LIN {X 0,Y 466.782,Z 446.473,A -85,B 0,C 180,E1 -7483.052,E2 -7483.052} C_VEL
LIN {X 0,Y 466.617,Z 450.017,A -85,B 0,C 180,E1 -7484.835,E2 -7484.835} C_VEL
LIN {X 0,Y 466.515,Z 452.31,A -85,B 0,C 180,E1 -7486.632,E2 -7486.632} C_VEL
LIN {X 0,Y 466.556,Z 453.367,A -85,B 0,C 180,E1 -7488.441,E2 -7488.441} C_VEL
LIN {X 0,Y 466.556,Z 453.179,A -85,B 0,C 180,E1 -7490.271,E2 -7490.271} C_VEL
LIN {X 0,Y 466.538,Z 451.697,A -85,B 0,C 180,E1 -7492.123,E2 -7492.123} C_VEL
LIN {X 0,Y 466.702,Z 448.846,A -85,B 0,C 180,E1 -7493.99,E2 -7493.99} C_VEL
LIN {X 0,Y 466.897,Z 444.505,A -85,B 0,C 180,E1 -7495.882,E2 -7495.882} C_VEL
LIN {X 0,Y 467.049,Z 439.911,A -85,B 0,C 180,E1 -7497.399,E2 -7497.399} C_VEL
LIN {X 0,Y 467.44,Z 432.616,A -85,B 0,C 180,E1 -7499.303,E2 -7499.303} C_VEL
LIN {X 0,Y 467.943,Z 424.827,A -85,B 0,C 180,E1 -7500.924,E2 -7500.924} C_VEL
LIN {X 0,Y 468.484,Z 416.084,A -85,B 0,C 180,E1 -7502.432,E2 -7502.432} C_VEL
LIN {X 0,Y 469.232,Z 405.809,A -85,B 0,C 180,E1 -7503.912,E2 -7503.912} C_VEL
LIN {X 0,Y 469.994,Z 394.444,A -85,B 0,C 180,E1 -7505.28,E2 -7505.28} C_VEL
LIN {X 0,Y 470.915,Z 381.942,A -85,B 0,C 180,E1 -7506.527,E2 -7506.527} C_VEL
LIN {X 0,Y 471.73,Z 369.989,A -85,B 0,C 180,E1 -7507.515,E2 -7507.515} C_VEL
LIN {X 0,Y 472.515,Z 356.993,A -85,B 0,C 180,E1 -7508.405,E2 -7508.405} C_VEL
LIN {X 0,Y 473.293,Z 342.587,A -85,B 0,C 180,E1 -7509.192,E2 -7509.192} C_VEL
LIN {X 0,Y 473.911,Z 327.391,A -85,B 0,C 180,E1 -7509.826,E2 -7509.826} C_VEL
LIN {X 0,Y 474.427,Z 311.981,A -85,B 0,C 180,E1 -7510.276,E2 -7510.276} C_VEL
LIN {X 0,Y 474.73,Z 291.402,A -85,B 0,C 180,E1 -7510.646,E2 -7510.646} C_VEL
LIN {X 0,Y 476.309,Z 163.823,A -85,B 0,C 180,E1 -7512.654,E2 -7512.654} C_VEL
LIN {X 0,Y 472.095,Z 146.225,A -85,B 0,C 180,E1 -7513.196,E2 -7513.196} C_VEL
LIN {X 0,Y 471.241,Z 143.803,A -85,B 0,C 180,E1 -7513.317,E2 -7513.317} C_VEL
LIN {X 0,Y 468.712,Z 132.548,A -85,B 0,C 180,E1 -7515.49,E2 -7515.49} C_VEL
LIN {X 0,Y 467.569,Z 127.869,A -85,B 0,C 180,E1 -7516.442,E2 -7516.442} C_VEL
LIN {X 0,Y 467.571,Z 127.872,A -85,B 0,C 180,E1 -7519.734,E2 -7519.734} C_VEL
LIN {X 0,Y 467.544,Z 127.872,A -85,B 0,C 180,E1 -7522.814,E2 -7522.814} C_VEL
LIN {X 0,Y 467.588,Z 127.867,A -85,B 0,C 180,E1 -7526.211,E2 -7526.211} C_VEL
LIN {X 0,Y 467.57,Z 127.865,A -85,B 0,C 180,E1 -7529.266,E2 -7529.266} C_VEL
LIN {X 0,Y 467.605,Z 127.861,A -85,B 0,C 180,E1 -7532.468,E2 -7532.468} C_VEL
LIN {X 0,Y 467.569,Z 127.862,A -85,B 0,C 180,E1 -7535.11,E2 -7535.11} C_VEL
LIN {X 0,Y 467.536,Z 127.873,A -85,B 0,C 180,E1 -7537.926,E2 -7537.926} C_VEL
LIN {X 0,Y 467.622,Z 127.859,A -85,B 0,C 180,E1 -7540.692,E2 -7540.692} C_VEL
LIN {X 0,Y 467.639,Z 127.856,A -85,B 0,C 180,E1 -7544.305,E2 -7544.305} C_VEL
LIN {X 0,Y 467.657,Z 127.855,A -85,B 0,C 180,E1 -7547.854,E2 -7547.854} C_VEL
LIN {X 0,Y 467.681,Z 127.852,A -85,B 0,C 180,E1 -7551.357,E2 -7551.357} C_VEL
LIN {X 0,Y 467.735,Z 127.842,A -85,B 0,C 180,E1 -7553.962,E2 -7553.962} C_VEL
LIN {X 0,Y 467.859,Z 127.831,A -85,B 0,C 180,E1 -7557.417,E2 -7557.417} C_VEL
LIN {X 0,Y 467.883,Z 127.826,A -85,B 0,C 180,E1 -7560,E2 -7560} C_VEL
LIN {X 0,Y 467.859,Z 127.827,A -85,B 0,C 180,E1 -7562.583,E2 -7562.583} C_VEL
LIN {X 0,Y 467.724,Z 127.844,A -85,B 0,C 180,E1 -7566.037,E2 -7566.037} C_VEL
LIN {X 0,Y 467.659,Z 127.856,A -85,B 0,C 180,E1 -7569.515,E2 -7569.515} C_VEL
LIN {X 0,Y 467.654,Z 127.852,A -85,B 0,C 180,E1 -7572.357,E2 -7572.357} C_VEL
LIN {X 0,Y 467.649,Z 127.85,A -85,B 0,C 180,E1 -7575.885,E2 -7575.885} C_VEL
LIN {X 0,Y 467.621,Z 127.857,A -85,B 0,C 180,E1 -7579.308,E2 -7579.308} C_VEL
LIN {X 0,Y 467.534,Z 127.869,A -85,B 0,C 180,E1 -7582.074,E2 -7582.074} C_VEL
LIN {X 0,Y 467.594,Z 127.866,A -85,B 0,C 180,E1 -7584.888,E2 -7584.888} C_VEL
LIN {X 0,Y 467.619,Z 127.859,A -85,B 0,C 180,E1 -7587.769,E2 -7587.769} C_VEL
LIN {X 0,Y 467.567,Z 127.866,A -85,B 0,C 180,E1 -7591.045,E2 -7591.045} C_VEL
LIN {X 0,Y 467.575,Z 127.868,A -85,B 0,C 180,E1 -7594.24,E2 -7594.24} C_VEL
LIN {X 0,Y 467.546,Z 127.866,A -85,B 0,C 180,E1 -7597.186,E2 -7597.186} C_VEL
LIN {X 0,Y 467.573,Z 127.866,A -85,B 0,C 180,E1 -7600.265,E2 -7600.265} C_VEL
LIN {X 0,Y 467.585,Z 127.858,A -85,B 0,C 180,E1 -7602.567,E2 -7602.567} C_VEL
LIN {X 0,Y 467.569,Z 127.866,A -85,B 0,C 180,E1 -7605.053,E2 -7605.053} C_VEL
LIN {X 0,Y 467.587,Z 127.86,A -85,B 0,C 180,E1 -7607.44,E2 -7607.44} C_VEL
LIN {X 0,Y 467.581,Z 127.866,A -85,B 0,C 180,E1 -7610.855,E2 -7610.855} C_VEL
LIN {X 0,Y 467.558,Z 127.87,A -85,B 0,C 180,E1 -7614.261,E2 -7614.261} C_VEL
LIN {X 0,Y 467.58,Z 127.863,A -85,B 0,C 180,E1 -7617.321,E2 -7617.321} C_VEL
LIN {X 0,Y 467.597,Z 127.89,A -85,B 0,C 180,E1 -7619.394,E2 -7619.394} C_VEL
LIN {X 0,Y 471.135,Z 142.057,A -85,B 0,C 180,E1 -7621.918,E2 -7621.918} C_VEL
LIN {X 0,Y 472.352,Z 148.297,A -85,B 0,C 180,E1 -7622.972,E2 -7622.972} C_VEL
LIN {X 0,Y 471.282,Z 166.846,A -85,B 0,C 180,E1 -7625.75,E2 -7625.75} C_VEL
LIN {X 0,Y 476.101,Z 191.193,A -85,B 0,C 180,E1 -7626.44,E2 -7626.44} C_VEL
LIN {X 0,Y 474.313,Z 333.167,A -85,B 0,C 180,E1 -7628.686,E2 -7628.686} C_VEL
LIN {X 0,Y 473.716,Z 349.25,A -85,B 0,C 180,E1 -7629.113,E2 -7629.113} C_VEL
LIN {X 0,Y 473.056,Z 364.395,A -85,B 0,C 180,E1 -7629.704,E2 -7629.704} C_VEL
LIN {X 0,Y 472.265,Z 378.653,A -85,B 0,C 180,E1 -7630.438,E2 -7630.438} C_VEL
LIN {X 0,Y 471.44,Z 392.03,A -85,B 0,C 180,E1 -7631.306,E2 -7631.306} C_VEL
LIN {X 0,Y 470.527,Z 405.676,A -85,B 0,C 180,E1 -7632.395,E2 -7632.395} C_VEL
LIN {X 0,Y 469.658,Z 418.059,A -85,B 0,C 180,E1 -7633.594,E2 -7633.594} C_VEL
LIN {X 0,Y 468.795,Z 430.236,A -85,B 0,C 180,E1 -7635.013,E2 -7635.013} C_VEL
LIN {X 0,Y 468.095,Z 441.083,A -85,B 0,C 180,E1 -7636.543,E2 -7636.543} C_VEL
LIN {X 0,Y 467.588,Z 450.127,A -85,B 0,C 180,E1 -7638.073,E2 -7638.073} C_VEL
LIN {X 0,Y 467.221,Z 457.636,A -85,B 0,C 180,E1 -7639.601,E2 -7639.601} C_VEL
LIN {X 0,Y 466.904,Z 464.643,A -85,B 0,C 180,E1 -7641.343,E2 -7641.343} C_VEL
LIN {X 0,Y 466.742,Z 470.157,A -85,B 0,C 180,E1 -7643.082,E2 -7643.082} C_VEL
LIN {X 0,Y 466.684,Z 474.33,A -85,B 0,C 180,E1 -7644.816,E2 -7644.816} C_VEL
LIN {X 0,Y 466.634,Z 477.256,A -85,B 0,C 180,E1 -7646.546,E2 -7646.546} C_VEL
LIN {X 0,Y 466.604,Z 479.003,A -85,B 0,C 180,E1 -7648.274,E2 -7648.274} C_VEL
LIN {X 0,Y 466.596,Z 479.604,A -85,B 0,C 180,E1 -7650,E2 -7650} C_VEL
LIN {X 0,Y 466.604,Z 479.005,A -85,B 0,C 180,E1 -7651.727,E2 -7651.727} C_VEL
LIN {X 0,Y 466.634,Z 477.252,A -85,B 0,C 180,E1 -7653.454,E2 -7653.454} C_VEL
LIN {X 0,Y 466.686,Z 474.32,A -85,B 0,C 180,E1 -7655.184,E2 -7655.184} C_VEL
LIN {X 0,Y 466.818,Z 470.137,A -85,B 0,C 180,E1 -7656.918,E2 -7656.918} C_VEL
LIN {X 0,Y 466.906,Z 464.586,A -85,B 0,C 180,E1 -7658.658,E2 -7658.658} C_VEL
LIN {X 0,Y 467.225,Z 457.523,A -85,B 0,C 180,E1 -7660.4,E2 -7660.4} C_VEL
LIN {X 0,Y 467.608,Z 449.968,A -85,B 0,C 180,E1 -7661.927,E2 -7661.927} C_VEL
LIN {X 0,Y 468.072,Z 440.853,A -85,B 0,C 180,E1 -7663.458,E2 -7663.458} C_VEL
LIN {X 0,Y 468.787,Z 429.87,A -85,B 0,C 180,E1 -7664.988,E2 -7664.988} C_VEL
LIN {X 0,Y 469.549,Z 418.573,A -85,B 0,C 180,E1 -7666.299,E2 -7666.299} C_VEL
LIN {X 0,Y 470.358,Z 406.169,A -85,B 0,C 180,E1 -7667.5,E2 -7667.5} C_VEL
LIN {X 0,Y 471.26,Z 392.481,A -85,B 0,C 180,E1 -7668.589,E2 -7668.589} C_VEL
LIN {X 0,Y 472.067,Z 379.034,A -85,B 0,C 180,E1 -7669.458,E2 -7669.458} C_VEL
LIN {X 0,Y 472.869,Z 364.303,A -85,B 0,C 180,E1 -7670.212,E2 -7670.212} C_VEL
LIN {X 0,Y 473.486,Z 349.003,A -85,B 0,C 180,E1 -7670.8,E2 -7670.8} C_VEL
LIN {X 0,Y 473.96,Z 333.066,A -85,B 0,C 180,E1 -7671.218,E2 -7671.218} C_VEL
LIN {X 0,Y 475.74,Z 191.939,A -85,B 0,C 180,E1 -7673.418,E2 -7673.418} C_VEL
LIN {X 0,Y 471.033,Z 167.135,A -85,B 0,C 180,E1 -7674.068,E2 -7674.068} C_VEL
LIN {X 0,Y 472.031,Z 148.627,A -85,B 0,C 180,E1 -7676.782,E2 -7676.782} C_VEL
LIN {X 0,Y 471.422,Z 143.906,A -85,B 0,C 180,E1 -7677.526,E2 -7677.526} C_VEL
LIN {X 0,Y 467.57,Z 127.869,A -85,B 0,C 180,E1 -7680.235,E2 -7680.235} C_VEL
LIN {X 0,Y 467.585,Z 127.868,A -85,B 0,C 180,E1 -7682.759,E2 -7682.759} C_VEL
LIN {X 0,Y 467.555,Z 127.873,A -85,B 0,C 180,E1 -7685.89,E2 -7685.89} C_VEL
LIN {X 0,Y 467.56,Z 127.867,A -85,B 0,C 180,E1 -7689.148,E2 -7689.148} C_VEL
LIN {X 0,Y 467.575,Z 127.868,A -85,B 0,C 180,E1 -7691.404,E2 -7691.404} C_VEL
LIN {X 0,Y 467.568,Z 127.868,A -85,B 0,C 180,E1 -7695.053,E2 -7695.053} C_VEL
LIN {X 0,Y 467.591,Z 127.87,A -85,B 0,C 180,E1 -7697.44,E2 -7697.44} C_VEL
LIN {X 0,Y 467.561,Z 127.864,A -85,B 0,C 180,E1 -7700.853,E2 -7700.853} C_VEL
LIN {X 0,Y 467.562,Z 127.864,A -85,B 0,C 180,E1 -7704.262,E2 -7704.262} C_VEL
LIN {X 0,Y 467.582,Z 127.867,A -85,B 0,C 180,E1 -7707.322,E2 -7707.322} C_VEL
LIN {X 0,Y 467.545,Z 127.865,A -85,B 0,C 180,E1 -7710.262,E2 -7710.262} C_VEL
LIN {X 0,Y 467.566,Z 127.86,A -85,B 0,C 180,E1 -7713.197,E2 -7713.197} C_VEL
LIN {X 0,Y 467.593,Z 127.862,A -85,B 0,C 180,E1 -7716.47,E2 -7716.47} C_VEL
LIN {X 0,Y 467.625,Z 127.856,A -85,B 0,C 180,E1 -7719.778,E2 -7719.778} C_VEL
LIN {X 0,Y 467.597,Z 127.864,A -85,B 0,C 180,E1 -7722.507,E2 -7722.507} C_VEL
LIN {X 0,Y 467.6,Z 127.862,A -85,B 0,C 180,E1 -7725.197,E2 -7725.197} C_VEL
LIN {X 0,Y 467.661,Z 127.85,A -85,B 0,C 180,E1 -7727.855,E2 -7727.855} C_VEL
LIN {X 0,Y 467.668,Z 127.85,A -85,B 0,C 180,E1 -7731.357,E2 -7731.357} C_VEL
LIN {X 0,Y 467.706,Z 127.848,A -85,B 0,C 180,E1 -7733.962,E2 -7733.962} C_VEL
LIN {X 0,Y 467.817,Z 127.828,A -85,B 0,C 180,E1 -7737.417,E2 -7737.417} C_VEL
LIN {X 0,Y 467.853,Z 127.817,A -85,B 0,C 180,E1 -7740,E2 -7740} C_VEL
LIN {X 0,Y 467.815,Z 127.833,A -85,B 0,C 180,E1 -7742.584,E2 -7742.584} C_VEL
LIN {X 0,Y 467.705,Z 127.85,A -85,B 0,C 180,E1 -7746.038,E2 -7746.038} C_VEL
LIN {X 0,Y 467.634,Z 127.842,A -85,B 0,C 180,E1 -7748.644,E2 -7748.644} C_VEL
LIN {X 0,Y 467.646,Z 127.855,A -85,B 0,C 180,E1 -7752.146,E2 -7752.146} C_VEL
LIN {X 0,Y 467.582,Z 127.867,A -85,B 0,C 180,E1 -7755.697,E2 -7755.697} C_VEL
LIN {X 0,Y 467.553,Z 127.865,A -85,B 0,C 180,E1 -7758.739,E2 -7758.739} C_VEL
LIN {X 0,Y 467.517,Z 127.869,A -85,B 0,C 180,E1 -7762.075,E2 -7762.075} C_VEL
LIN {X 0,Y 467.531,Z 127.87,A -85,B 0,C 180,E1 -7764.892,E2 -7764.892} C_VEL
LIN {X 0,Y 467.542,Z 127.86,A -85,B 0,C 180,E1 -7767.775,E2 -7767.775} C_VEL
LIN {X 0,Y 467.532,Z 127.862,A -85,B 0,C 180,E1 -7771.036,E2 -7771.036} C_VEL
LIN {X 0,Y 467.568,Z 127.863,A -85,B 0,C 180,E1 -7774.238,E2 -7774.238} C_VEL
LIN {X 0,Y 467.518,Z 127.863,A -85,B 0,C 180,E1 -7777.181,E2 -7777.181} C_VEL
LIN {X 0,Y 467.561,Z 127.861,A -85,B 0,C 180,E1 -7780.267,E2 -7780.267} C_VEL
LIN {X 0,Y 467.55,Z 127.864,A -85,B 0,C 180,E1 -7783.746,E2 -7783.746} C_VEL
LIN {X 0,Y 467.55,Z 127.857,A -85,B 0,C 180,E1 -7786.254,E2 -7786.254} C_VEL
LIN {X 0,Y 467.561,Z 127.865,A -85,B 0,C 180,E1 -7789.733,E2 -7789.733} C_VEL
LIN {X 0,Y 467.526,Z 127.869,A -85,B 0,C 180,E1 -7793.037,E2 -7793.037} C_VEL
LIN {X 0,Y 467.573,Z 127.868,A -85,B 0,C 180,E1 -7796.21,E2 -7796.21} C_VEL
LIN {X 0,Y 467.571,Z 127.865,A -85,B 0,C 180,E1 -7799.266,E2 -7799.266} C_VEL
LIN {X 0,Y 467.556,Z 127.872,A -85,B 0,C 180,E1 -7802.481,E2 -7802.481} C_VEL
LIN {X 0,Y 467.565,Z 127.867,A -85,B 0,C 180,E1 -7805.11,E2 -7805.11} C_VEL
LIN {X 0,Y 467.54,Z 127.874,A -85,B 0,C 180,E1 -7807.926,E2 -7807.926} C_VEL
LIN {X 0,Y 467.626,Z 127.856,A -85,B 0,C 180,E1 -7810.692,E2 -7810.692} C_VEL
LIN {X 0,Y 467.644,Z 127.859,A -85,B 0,C 180,E1 -7814.305,E2 -7814.305} C_VEL
LIN {X 0,Y 467.598,Z 127.861,A -85,B 0,C 180,E1 -7815.378,E2 -7815.378} C_VEL
LIN {X 0,Y 466.926,Z 127.942,A -85,B 0,C 180,E1 -7816.097,E2 -7816.097} C_VEL
LIN {X 0,Y 464.087,Z 128.299,A -85,B 0,C 180,E1 -7817.265,E2 -7817.265} C_VEL
LIN {X 0,Y 461.69,Z 128.601,A -85,B 0,C 180,E1 -7818.208,E2 -7818.208} C_VEL
LIN {X 0,Y 460.662,Z 128.729,A -85,B 0,C 180,E1 -7818.936,E2 -7818.936} C_VEL
LIN {X 0,Y 460.578,Z 128.74,A -85,B 0,C 180,E1 -7819.182,E2 -7819.182} C_VEL
LIN {X 0,Y 460.666,Z 128.88,A -85,B 0,C 180,E1 -7821.832,E2 -7821.832} C_VEL
LIN {X 0,Y 463.902,Z 143.363,A -85,B 0,C 180,E1 -7824.566,E2 -7824.566} C_VEL
LIN {X 0,Y 463.975,Z 143.816,A -85,B 0,C 180,E1 -7824.649,E2 -7824.649} C_VEL
LIN {X 0,Y 465.945,Z 150.272,A -85,B 0,C 180,E1 -7824.861,E2 -7824.861} C_VEL
LIN {X 0,Y 469.269,Z 165.031,A -85,B 0,C 180,E1 -7825.274,E2 -7825.274} C_VEL
LIN {X 0,Y 467.513,Z 308.285,A -85,B 0,C 180,E1 -7827.55,E2 -7827.55} C_VEL
LIN {X 0,Y 467.068,Z 323.449,A -85,B 0,C 180,E1 -7827.952,E2 -7827.952} C_VEL
LIN {X 0,Y 466.484,Z 338.755,A -85,B 0,C 180,E1 -7828.543,E2 -7828.543} C_VEL
LIN {X 0,Y 465.789,Z 352.417,A -85,B 0,C 180,E1 -7829.243,E2 -7829.243} C_VEL
LIN {X 0,Y 464.987,Z 365.876,A -85,B 0,C 180,E1 -7830.108,E2 -7830.108} C_VEL
LIN {X 0,Y 464.087,Z 378.978,A -85,B 0,C 180,E1 -7831.141,E2 -7831.141} C_VEL
LIN {X 0,Y 463.273,Z 390.919,A -85,B 0,C 180,E1 -7832.282,E2 -7832.282} C_VEL
LIN {X 0,Y 462.469,Z 401.527,A -85,B 0,C 180,E1 -7833.485,E2 -7833.485} C_VEL
LIN {X 0,Y 461.736,Z 411.376,A -85,B 0,C 180,E1 -7834.802,E2 -7834.802} C_VEL
LIN {X 0,Y 461.14,Z 421.006,A -85,B 0,C 180,E1 -7836.343,E2 -7836.343} C_VEL
LIN {X 0,Y 460.609,Z 429.084,A -85,B 0,C 180,E1 -7837.893,E2 -7837.893} C_VEL
LIN {X 0,Y 460.133,Z 436.655,A -85,B 0,C 180,E1 -7839.672,E2 -7839.672} C_VEL
LIN {X 0,Y 459.858,Z 442.694,A -85,B 0,C 180,E1 -7841.459,E2 -7841.459} C_VEL
LIN {X 0,Y 459.664,Z 447.348,A -85,B 0,C 180,E1 -7843.258,E2 -7843.258} C_VEL
LIN {X 0,Y 459.528,Z 450.686,A -85,B 0,C 180,E1 -7845.07,E2 -7845.07} C_VEL
LIN {X 0,Y 459.429,Z 452.771,A -85,B 0,C 180,E1 -7846.896,E2 -7846.896} C_VEL
LIN {X 0,Y 459.443,Z 453.621,A -85,B 0,C 180,E1 -7848.737,E2 -7848.737} C_VEL
LIN {X 0,Y 459.449,Z 453.22,A -85,B 0,C 180,E1 -7850.598,E2 -7850.598} C_VEL
LIN {X 0,Y 459.464,Z 451.518,A -85,B 0,C 180,E1 -7852.482,E2 -7852.482} C_VEL
LIN {X 0,Y 459.645,Z 448.435,A -85,B 0,C 180,E1 -7854.383,E2 -7854.383} C_VEL
LIN {X 0,Y 459.862,Z 443.845,A -85,B 0,C 180,E1 -7856.308,E2 -7856.308} C_VEL
LIN {X 0,Y 460.067,Z 438.9,A -85,B 0,C 180,E1 -7857.895,E2 -7857.895} C_VEL
LIN {X 0,Y 460.456,Z 432.522,A -85,B 0,C 180,E1 -7859.54,E2 -7859.54} C_VEL
LIN {X 0,Y 461.008,Z 424.517,A -85,B 0,C 180,E1 -7861.22,E2 -7861.22} C_VEL
LIN {X 0,Y 461.591,Z 415.894,A -85,B 0,C 180,E1 -7862.718,E2 -7862.718} C_VEL
LIN {X 0,Y 462.397,Z 405.555,A -85,B 0,C 180,E1 -7864.219,E2 -7864.219} C_VEL
LIN {X 0,Y 463.258,Z 394.112,A -85,B 0,C 180,E1 -7865.604,E2 -7865.604} C_VEL
LIN {X 0,Y 464.244,Z 381.493,A -85,B 0,C 180,E1 -7866.868,E2 -7866.868} C_VEL
LIN {X 0,Y 465.203,Z 367.754,A -85,B 0,C 180,E1 -7867.997,E2 -7867.997} C_VEL
LIN {X 0,Y 466.106,Z 353.975,A -85,B 0,C 180,E1 -7868.91,E2 -7868.91} C_VEL
LIN {X 0,Y 466.896,Z 339.006,A -85,B 0,C 180,E1 -7869.69,E2 -7869.69} C_VEL
LIN {X 0,Y 467.472,Z 324.137,A -85,B 0,C 180,E1 -7870.275,E2 -7870.275} C_VEL
LIN {X 0,Y 468.003,Z 308.311,A -85,B 0,C 180,E1 -7870.697,E2 -7870.697} C_VEL
LIN {X 0,Y 469.919,Z 165.105,A -85,B 0,C 180,E1 -7873.005,E2 -7873.005} C_VEL
LIN {X 0,Y 466.02,Z 148.879,A -85,B 0,C 180,E1 -7873.518,E2 -7873.518} C_VEL
LIN {X 0,Y 464.143,Z 144.12,A -85,B 0,C 180,E1 -7873.733,E2 -7873.733} C_VEL
LIN {X 0,Y 461.347,Z 132.074,A -85,B 0,C 180,E1 -7876.121,E2 -7876.121} C_VEL
LIN {X 0,Y 460.54,Z 128.745,A -85,B 0,C 180,E1 -7876.816,E2 -7876.816} C_VEL
LIN {X 0,Y 460.52,Z 128.748,A -85,B 0,C 180,E1 -7880.136,E2 -7880.136} C_VEL
LIN {X 0,Y 460.474,Z 128.752,A -85,B 0,C 180,E1 -7883.47,E2 -7883.47} C_VEL
LIN {X 0,Y 460.531,Z 128.744,A -85,B 0,C 180,E1 -7886.675,E2 -7886.675} C_VEL
LIN {X 0,Y 460.508,Z 128.747,A -85,B 0,C 180,E1 -7889.759,E2 -7889.759} C_VEL
LIN {X 0,Y 460.535,Z 128.741,A -85,B 0,C 180,E1 -7892.753,E2 -7892.753} C_VEL
LIN {X 0,Y 460.522,Z 128.738,A -85,B 0,C 180,E1 -7895.666,E2 -7895.666} C_VEL
LIN {X 0,Y 460.523,Z 128.743,A -85,B 0,C 180,E1 -7898.578,E2 -7898.578} C_VEL
LIN {X 0,Y 460.586,Z 128.737,A -85,B 0,C 180,E1 -7901.31,E2 -7901.31} C_VEL
LIN {X 0,Y 460.605,Z 128.734,A -85,B 0,C 180,E1 -7904.059,E2 -7904.059} C_VEL
LIN {X 0,Y 460.61,Z 128.734,A -85,B 0,C 180,E1 -7907.665,E2 -7907.665} C_VEL
LIN {X 0,Y 460.628,Z 128.73,A -85,B 0,C 180,E1 -7911.223,E2 -7911.223} C_VEL
LIN {X 0,Y 460.701,Z 128.719,A -85,B 0,C 180,E1 -7913.87,E2 -7913.87} C_VEL
LIN {X 0,Y 460.799,Z 128.711,A -85,B 0,C 180,E1 -7917.377,E2 -7917.377} C_VEL
LIN {X 0,Y 460.853,Z 128.702,A -85,B 0,C 180,E1 -7920,E2 -7920} C_VEL
LIN {X 0,Y 460.8,Z 128.706,A -85,B 0,C 180,E1 -7922.622,E2 -7922.622} C_VEL
LIN {X 0,Y 460.688,Z 128.721,A -85,B 0,C 180,E1 -7926.13,E2 -7926.13} C_VEL
LIN {X 0,Y 460.619,Z 128.731,A -85,B 0,C 180,E1 -7928.776,E2 -7928.776} C_VEL
LIN {X 0,Y 460.613,Z 128.729,A -85,B 0,C 180,E1 -7932.445,E2 -7932.445} C_VEL
LIN {X 0,Y 460.6,Z 128.728,A -85,B 0,C 180,E1 -7935.997,E2 -7935.997} C_VEL
LIN {X 0,Y 460.567,Z 128.734,A -85,B 0,C 180,E1 -7939.615,E2 -7939.615} C_VEL
LIN {X 0,Y 460.51,Z 128.747,A -85,B 0,C 180,E1 -7942.428,E2 -7942.428} C_VEL
LIN {X 0,Y 460.557,Z 128.736,A -85,B 0,C 180,E1 -7945.799,E2 -7945.799} C_VEL
LIN {X 0,Y 460.551,Z 128.742,A -85,B 0,C 180,E1 -7948.233,E2 -7948.233} C_VEL
LIN {X 0,Y 460.519,Z 128.743,A -85,B 0,C 180,E1 -7951.283,E2 -7951.283} C_VEL
LIN {X 0,Y 460.521,Z 128.746,A -85,B 0,C 180,E1 -7954.504,E2 -7954.504} C_VEL
LIN {X 0,Y 460.499,Z 128.743,A -85,B 0,C 180,E1 -7957.623,E2 -7957.623} C_VEL
LIN {X 0,Y 460.537,Z 128.742,A -85,B 0,C 180,E1 -7960.269,E2 -7960.269} C_VEL
LIN {X 0,Y 460.498,Z 128.738,A -85,B 0,C 180,E1 -7963.375,E2 -7963.375} C_VEL
LIN {X 0,Y 460.498,Z 128.742,A -85,B 0,C 180,E1 -7966.625,E2 -7966.625} C_VEL
LIN {X 0,Y 460.54,Z 128.74,A -85,B 0,C 180,E1 -7969.731,E2 -7969.731} C_VEL
LIN {X 0,Y 460.498,Z 128.745,A -85,B 0,C 180,E1 -7972.524,E2 -7972.524} C_VEL
LIN {X 0,Y 460.545,Z 128.741,A -85,B 0,C 180,E1 -7975.624,E2 -7975.624} C_VEL
LIN {X 0,Y 460.531,Z 128.762,A -85,B 0,C 180,E1 -7979,E2 -7979} C_VEL
LIN {X 0,Y 463.991,Z 142.229,A -85,B 0,C 180,E1 -7981.464,E2 -7981.464} C_VEL
LIN {X 0,Y 465.574,Z 150.285,A -85,B 0,C 180,E1 -7982.855,E2 -7982.855} C_VEL
LIN {X 0,Y 464.571,Z 166.588,A -85,B 0,C 180,E1 -7985.338,E2 -7985.338} C_VEL
LIN {X 0,Y 469.673,Z 192.497,A -85,B 0,C 180,E1 -7986.096,E2 -7986.096} C_VEL
LIN {X 0,Y 467.74,Z 333.751,A -85,B 0,C 180,E1 -7988.371,E2 -7988.371} C_VEL
LIN {X 0,Y 467.106,Z 349.529,A -85,B 0,C 180,E1 -7988.804,E2 -7988.804} C_VEL
LIN {X 0,Y 466.384,Z 364.91,A -85,B 0,C 180,E1 -7989.42,E2 -7989.42} C_VEL
LIN {X 0,Y 465.583,Z 378.735,A -85,B 0,C 180,E1 -7990.145,E2 -7990.145} C_VEL
LIN {X 0,Y 464.691,Z 392.073,A -85,B 0,C 180,E1 -7991.025,E2 -7991.025} C_VEL
LIN {X 0,Y 463.717,Z 405.668,A -85,B 0,C 180,E1 -7992.127,E2 -7992.127} C_VEL
LIN {X 0,Y 462.8,Z 418.02,A -85,B 0,C 180,E1 -7993.344,E2 -7993.344} C_VEL
LIN {X 0,Y 461.887,Z 430.143,A -85,B 0,C 180,E1 -7994.783,E2 -7994.783} C_VEL
LIN {X 0,Y 461.113,Z 440.953,A -85,B 0,C 180,E1 -7996.335,E2 -7996.335} C_VEL
LIN {X 0,Y 460.571,Z 449.974,A -85,B 0,C 180,E1 -7997.889,E2 -7997.889} C_VEL
LIN {X 0,Y 460.208,Z 457.479,A -85,B 0,C 180,E1 -7999.441,E2 -7999.441} C_VEL
LIN {X 0,Y 459.847,Z 464.478,A -85,B 0,C 180,E1 -8001.209,E2 -8001.209} C_VEL
LIN {X 0,Y 459.662,Z 469.985,A -85,B 0,C 180,E1 -8002.975,E2 -8002.975} C_VEL
LIN {X 0,Y 459.595,Z 474.15,A -85,B 0,C 180,E1 -8004.736,E2 -8004.736} C_VEL
LIN {X 0,Y 459.529,Z 477.07,A -85,B 0,C 180,E1 -8006.493,E2 -8006.493} C_VEL
LIN {X 0,Y 459.517,Z 478.81,A -85,B 0,C 180,E1 -8008.247,E2 -8008.247} C_VEL
LIN {X 0,Y 459.527,Z 479.405,A -85,B 0,C 180,E1 -8010,E2 -8010} C_VEL
LIN {X 0,Y 459.517,Z 478.8,A -85,B 0,C 180,E1 -8011.753,E2 -8011.753} C_VEL
LIN {X 0,Y 459.53,Z 477.038,A -85,B 0,C 180,E1 -8013.508,E2 -8013.508} C_VEL
LIN {X 0,Y 459.598,Z 474.096,A -85,B 0,C 180,E1 -8015.265,E2 -8015.265} C_VEL
LIN {X 0,Y 459.727,Z 469.902,A -85,B 0,C 180,E1 -8017.025,E2 -8017.025} C_VEL
LIN {X 0,Y 459.848,Z 464.339,A -85,B 0,C 180,E1 -8018.792,E2 -8018.792} C_VEL
LIN {X 0,Y 460.202,Z 457.264,A -85,B 0,C 180,E1 -8020.56,E2 -8020.56} C_VEL
LIN {X 0,Y 460.584,Z 449.695,A -85,B 0,C 180,E1 -8022.112,E2 -8022.112} C_VEL
LIN {X 0,Y 461.108,Z 440.568,A -85,B 0,C 180,E1 -8023.665,E2 -8023.665} C_VEL
LIN {X 0,Y 461.855,Z 429.56,A -85,B 0,C 180,E1 -8025.218,E2 -8025.218} C_VEL
LIN {X 0,Y 462.672,Z 418.234,A -85,B 0,C 180,E1 -8026.548,E2 -8026.548} C_VEL
LIN {X 0,Y 463.525,Z 405.778,A -85,B 0,C 180,E1 -8027.767,E2 -8027.767} C_VEL
LIN {X 0,Y 464.473,Z 392.009,A -85,B 0,C 180,E1 -8028.871,E2 -8028.871} C_VEL
LIN {X 0,Y 465.338,Z 378.488,A -85,B 0,C 180,E1 -8029.751,E2 -8029.751} C_VEL
LIN {X 0,Y 466.15,Z 364.121,A -85,B 0,C 180,E1 -8030.492,E2 -8030.492} C_VEL
LIN {X 0,Y 466.771,Z 349.319,A -85,B 0,C 180,E1 -8031.072,E2 -8031.072} C_VEL
LIN {X 0,Y 467.294,Z 333.178,A -85,B 0,C 180,E1 -8031.506,E2 -8031.506} C_VEL
LIN {X 0,Y 469.146,Z 192.736,A -85,B 0,C 180,E1 -8033.729,E2 -8033.729} C_VEL
LIN {X 0,Y 464.228,Z 166.936,A -85,B 0,C 180,E1 -8034.419,E2 -8034.419} C_VEL
LIN {X 0,Y 465.196,Z 149.867,A -85,B 0,C 180,E1 -8036.957,E2 -8036.957} C_VEL
LIN {X 0,Y 464.453,Z 145.092,A -85,B 0,C 180,E1 -8037.73,E2 -8037.73} C_VEL
LIN {X 0,Y 460.522,Z 128.748,A -85,B 0,C 180,E1 -8040.525,E2 -8040.525} C_VEL
LIN {X 0,Y 460.531,Z 128.748,A -85,B 0,C 180,E1 -8043.325,E2 -8043.325} C_VEL
LIN {X 0,Y 460.478,Z 128.753,A -85,B 0,C 180,E1 -8046.53,E2 -8046.53} C_VEL
LIN {X 0,Y 460.535,Z 128.742,A -85,B 0,C 180,E1 -8048.896,E2 -8048.896} C_VEL
LIN {X 0,Y 460.505,Z 128.747,A -85,B 0,C 180,E1 -8052.184,E2 -8052.184} C_VEL
LIN {X 0,Y 460.516,Z 128.751,A -85,B 0,C 180,E1 -8055.412,E2 -8055.412} C_VEL
LIN {X 0,Y 460.534,Z 128.743,A -85,B 0,C 180,E1 -8058.398,E2 -8058.398} C_VEL
LIN {X 0,Y 460.52,Z 128.742,A -85,B 0,C 180,E1 -8061.267,E2 -8061.267} C_VEL
LIN {X 0,Y 460.511,Z 128.742,A -85,B 0,C 180,E1 -8064.555,E2 -8064.555} C_VEL
LIN {X 0,Y 460.532,Z 128.742,A -85,B 0,C 180,E1 -8067.716,E2 -8067.716} C_VEL
LIN {X 0,Y 460.523,Z 128.743,A -85,B 0,C 180,E1 -8070.768,E2 -8070.768} C_VEL
LIN {X 0,Y 460.534,Z 128.735,A -85,B 0,C 180,E1 -8073.733,E2 -8073.733} C_VEL
LIN {X 0,Y 460.547,Z 128.742,A -85,B 0,C 180,E1 -8076.624,E2 -8076.624} C_VEL
LIN {X 0,Y 460.554,Z 128.738,A -85,B 0,C 180,E1 -8079.453,E2 -8079.453} C_VEL
LIN {X 0,Y 460.549,Z 128.739,A -85,B 0,C 180,E1 -8082.23,E2 -8082.23} C_VEL
LIN {X 0,Y 460.562,Z 128.741,A -85,B 0,C 180,E1 -8084.965,E2 -8084.965} C_VEL
LIN {X 0,Y 460.613,Z 128.734,A -85,B 0,C 180,E1 -8088.56,E2 -8088.56} C_VEL
LIN {X 0,Y 460.619,Z 128.728,A -85,B 0,C 180,E1 -8091.224,E2 -8091.224} C_VEL
LIN {X 0,Y 460.672,Z 128.723,A -85,B 0,C 180,E1 -8093.87,E2 -8093.87} C_VEL
LIN {X 0,Y 460.761,Z 128.707,A -85,B 0,C 180,E1 -8097.378,E2 -8097.378} C_VEL
LIN {X 0,Y 460.823,Z 128.692,A -85,B 0,C 180,E1 -8100,E2 -8100} C_VEL
LIN {X 0,Y 460.759,Z 128.712,A -85,B 0,C 180,E1 -8102.623,E2 -8102.623} C_VEL
LIN {X 0,Y 460.671,Z 128.724,A -85,B 0,C 180,E1 -8106.131,E2 -8106.131} C_VEL
LIN {X 0,Y 460.589,Z 128.718,A -85,B 0,C 180,E1 -8108.777,E2 -8108.777} C_VEL
LIN {X 0,Y 460.602,Z 128.73,A -85,B 0,C 180,E1 -8112.435,E2 -8112.435} C_VEL
LIN {X 0,Y 460.531,Z 128.741,A -85,B 0,C 180,E1 -8115.965,E2 -8115.965} C_VEL
LIN {X 0,Y 460.514,Z 128.742,A -85,B 0,C 180,E1 -8118.879,E2 -8118.879} C_VEL
LIN {X 0,Y 460.492,Z 128.742,A -85,B 0,C 180,E1 -8122.43,E2 -8122.43} C_VEL
LIN {X 0,Y 460.526,Z 128.742,A -85,B 0,C 180,E1 -8125.79,E2 -8125.79} C_VEL
LIN {X 0,Y 460.5,Z 128.734,A -85,B 0,C 180,E1 -8128.237,E2 -8128.237} C_VEL
LIN {X 0,Y 460.5,Z 128.741,A -85,B 0,C 180,E1 -8131.278,E2 -8131.278} C_VEL
LIN {X 0,Y 460.515,Z 128.743,A -85,B 0,C 180,E1 -8134.501,E2 -8134.501} C_VEL
LIN {X 0,Y 460.486,Z 128.734,A -85,B 0,C 180,E1 -8137.625,E2 -8137.625} C_VEL
LIN {X 0,Y 460.519,Z 128.747,A -85,B 0,C 180,E1 -8141.013,E2 -8141.013} C_VEL
LIN {X 0,Y 460.516,Z 128.743,A -85,B 0,C 180,E1 -8144.589,E2 -8144.589} C_VEL
LIN {X 0,Y 460.48,Z 128.745,A -85,B 0,C 180,E1 -8147.813,E2 -8147.813} C_VEL
LIN {X 0,Y 460.516,Z 128.745,A -85,B 0,C 180,E1 -8150.135,E2 -8150.135} C_VEL
LIN {X 0,Y 460.476,Z 128.745,A -85,B 0,C 180,E1 -8153.47,E2 -8153.47} C_VEL
LIN {X 0,Y 460.522,Z 128.74,A -85,B 0,C 180,E1 -8156.674,E2 -8156.674} C_VEL
LIN {X 0,Y 460.509,Z 128.746,A -85,B 0,C 180,E1 -8159.759,E2 -8159.759} C_VEL
LIN {X 0,Y 460.497,Z 128.749,A -85,B 0,C 180,E1 -8162.751,E2 -8162.751} C_VEL
LIN {X 0,Y 460.523,Z 128.746,A -85,B 0,C 180,E1 -8165.666,E2 -8165.666} C_VEL
LIN {X 0,Y 460.527,Z 128.744,A -85,B 0,C 180,E1 -8168.578,E2 -8168.578} C_VEL
LIN {X 0,Y 460.589,Z 128.733,A -85,B 0,C 180,E1 -8171.31,E2 -8171.31} C_VEL
LIN {X 0,Y 460.61,Z 128.738,A -85,B 0,C 180,E1 -8174.059,E2 -8174.059} C_VEL
LIN {X 0,Y 460.615,Z 128.736,A -85,B 0,C 180,E1 -8177.666,E2 -8177.666} C_VEL
LIN {X 0,Y 460.578,Z 128.74,A -85,B 0,C 180,E1 -8179.182,E2 -8179.182} C_VEL
LIN {X 0,Y 459.847,Z 128.893,A -85,B 0,C 180,E1 -8179.69,E2 -8179.69} C_VEL
LIN {X 0,Y 454.181,Z 129.586,A -85,B 0,C 180,E1 -8181.254,E2 -8181.254} C_VEL
LIN {X 0,Y 453.765,Z 130.303,A -85,B 0,C 180,E1 -8181.633,E2 -8181.633} C_VEL
LIN {X 0,Y 453.816,Z 130.602,A -85,B 0,C 180,E1 -8181.702,E2 -8181.702} C_VEL
LIN {X 0,Y 456.858,Z 144.007,A -85,B 0,C 180,E1 -8184.271,E2 -8184.271} C_VEL
LIN {X 0,Y 459.358,Z 151.363,A -85,B 0,C 180,E1 -8184.532,E2 -8184.532} C_VEL
LIN {X 0,Y 462.738,Z 166.534,A -85,B 0,C 180,E1 -8184.964,E2 -8184.964} C_VEL
LIN {X 0,Y 460.817,Z 309.517,A -85,B 0,C 180,E1 -8187.268,E2 -8187.268} C_VEL
LIN {X 0,Y 460.338,Z 325.111,A -85,B 0,C 180,E1 -8187.703,E2 -8187.703} C_VEL
LIN {X 0,Y 459.754,Z 339.99,A -85,B 0,C 180,E1 -8188.302,E2 -8188.302} C_VEL
LIN {X 0,Y 459.023,Z 353.474,A -85,B 0,C 180,E1 -8189.013,E2 -8189.013} C_VEL
LIN {X 0,Y 458.174,Z 366.768,A -85,B 0,C 180,E1 -8189.89,E2 -8189.89} C_VEL
LIN {X 0,Y 457.21,Z 380.349,A -85,B 0,C 180,E1 -8190.991,E2 -8190.991} C_VEL
LIN {X 0,Y 456.26,Z 392.664,A -85,B 0,C 180,E1 -8192.207,E2 -8192.207} C_VEL
LIN {X 0,Y 455.421,Z 403.883,A -85,B 0,C 180,E1 -8193.539,E2 -8193.539} C_VEL
LIN {X 0,Y 454.676,Z 413.378,A -85,B 0,C 180,E1 -8194.877,E2 -8194.877} C_VEL
LIN {X 0,Y 454.051,Z 422.718,A -85,B 0,C 180,E1 -8196.443,E2 -8196.443} C_VEL
LIN {X 0,Y 453.531,Z 430.532,A -85,B 0,C 180,E1 -8198.017,E2 -8198.017} C_VEL
LIN {X 0,Y 453.016,Z 437.873,A -85,B 0,C 180,E1 -8199.825,E2 -8199.825} C_VEL
LIN {X 0,Y 452.774,Z 443.682,A -85,B 0,C 180,E1 -8201.641,E2 -8201.641} C_VEL
LIN {X 0,Y 452.534,Z 448.128,A -85,B 0,C 180,E1 -8203.471,E2 -8203.471} C_VEL
LIN {X 0,Y 452.431,Z 451.282,A -85,B 0,C 180,E1 -8205.312,E2 -8205.312} C_VEL
LIN {X 0,Y 452.325,Z 453.205,A -85,B 0,C 180,E1 -8207.17,E2 -8207.17} C_VEL
LIN {X 0,Y 452.343,Z 453.875,A -85,B 0,C 180,E1 -8209.043,E2 -8209.043} C_VEL
LIN {X 0,Y 452.373,Z 453.262,A -85,B 0,C 180,E1 -8210.936,E2 -8210.936} C_VEL
LIN {X 0,Y 452.401,Z 451.34,A -85,B 0,C 180,E1 -8212.853,E2 -8212.853} C_VEL
LIN {X 0,Y 452.599,Z 448.027,A -85,B 0,C 180,E1 -8214.788,E2 -8214.788} C_VEL
LIN {X 0,Y 452.833,Z 443.195,A -85,B 0,C 180,E1 -8216.749,E2 -8216.749} C_VEL
LIN {X 0,Y 453.074,Z 438.432,A -85,B 0,C 180,E1 -8218.239,E2 -8218.239} C_VEL
LIN {X 0,Y 453.471,Z 432.46,A -85,B 0,C 180,E1 -8219.783,E2 -8219.783} C_VEL
LIN {X 0,Y 454.076,Z 424.621,A -85,B 0,C 180,E1 -8221.446,E2 -8221.446} C_VEL
LIN {X 0,Y 454.692,Z 415.928,A -85,B 0,C 180,E1 -8222.977,E2 -8222.977} C_VEL
LIN {X 0,Y 455.577,Z 405.298,A -85,B 0,C 180,E1 -8224.536,E2 -8224.536} C_VEL
LIN {X 0,Y 456.527,Z 393.767,A -85,B 0,C 180,E1 -8225.938,E2 -8225.938} C_VEL
LIN {X 0,Y 457.502,Z 381.555,A -85,B 0,C 180,E1 -8227.174,E2 -8227.174} C_VEL
LIN {X 0,Y 458.532,Z 367.84,A -85,B 0,C 180,E1 -8228.315,E2 -8228.315} C_VEL
LIN {X 0,Y 459.51,Z 353.755,A -85,B 0,C 180,E1 -8229.258,E2 -8229.258} C_VEL
LIN {X 0,Y 460.317,Z 339.35,A -85,B 0,C 180,E1 -8230.019,E2 -8230.019} C_VEL
LIN {X 0,Y 460.94,Z 324.627,A -85,B 0,C 180,E1 -8230.608,E2 -8230.608} C_VEL
LIN {X 0,Y 461.487,Z 308.491,A -85,B 0,C 180,E1 -8231.046,E2 -8231.046} C_VEL
LIN {X 0,Y 463.615,Z 167.212,A -85,B 0,C 180,E1 -8233.35,E2 -8233.35} C_VEL
LIN {X 0,Y 460.237,Z 152.305,A -85,B 0,C 180,E1 -8233.819,E2 -8233.819} C_VEL
LIN {X 0,Y 457.019,Z 144.383,A -85,B 0,C 180,E1 -8234.176,E2 -8234.176} C_VEL
LIN {X 0,Y 454.074,Z 132.104,A -85,B 0,C 180,E1 -8236.673,E2 -8236.673} C_VEL
LIN {X 0,Y 453.489,Z 129.627,A -85,B 0,C 180,E1 -8237.222,E2 -8237.222} C_VEL
LIN {X 0,Y 453.495,Z 129.626,A -85,B 0,C 180,E1 -8239.409,E2 -8239.409} C_VEL
LIN {X 0,Y 453.451,Z 129.627,A -85,B 0,C 180,E1 -8242.81,E2 -8242.81} C_VEL
LIN {X 0,Y 453.478,Z 129.622,A -85,B 0,C 180,E1 -8246.087,E2 -8246.087} C_VEL
LIN {X 0,Y 453.476,Z 129.62,A -85,B 0,C 180,E1 -8249.24,E2 -8249.24} C_VEL
LIN {X 0,Y 453.509,Z 129.614,A -85,B 0,C 180,E1 -8252.295,E2 -8252.295} C_VEL
LIN {X 0,Y 453.495,Z 129.616,A -85,B 0,C 180,E1 -8255.264,E2 -8255.264} C_VEL
LIN {X 0,Y 453.481,Z 129.622,A -85,B 0,C 180,E1 -8258.415,E2 -8258.415} C_VEL
LIN {X 0,Y 453.523,Z 129.615,A -85,B 0,C 180,E1 -8261.008,E2 -8261.008} C_VEL
LIN {X 0,Y 453.57,Z 129.613,A -85,B 0,C 180,E1 -8263.879,E2 -8263.879} C_VEL
LIN {X 0,Y 453.564,Z 129.613,A -85,B 0,C 180,E1 -8267.471,E2 -8267.471} C_VEL
LIN {X 0,Y 453.591,Z 129.606,A -85,B 0,C 180,E1 -8271.086,E2 -8271.086} C_VEL
LIN {X 0,Y 453.669,Z 129.596,A -85,B 0,C 180,E1 -8273.774,E2 -8273.774} C_VEL
LIN {X 0,Y 453.743,Z 129.59,A -85,B 0,C 180,E1 -8277.336,E2 -8277.336} C_VEL
LIN {X 0,Y 453.823,Z 129.578,A -85,B 0,C 180,E1 -8280,E2 -8280} C_VEL
LIN {X 0,Y 453.744,Z 129.586,A -85,B 0,C 180,E1 -8282.663,E2 -8282.663} C_VEL
LIN {X 0,Y 453.653,Z 129.597,A -85,B 0,C 180,E1 -8286.225,E2 -8286.225} C_VEL
LIN {X 0,Y 453.585,Z 129.607,A -85,B 0,C 180,E1 -8288.913,E2 -8288.913} C_VEL
LIN {X 0,Y 453.563,Z 129.608,A -85,B 0,C 180,E1 -8292.529,E2 -8292.529} C_VEL
LIN {X 0,Y 453.544,Z 129.608,A -85,B 0,C 180,E1 -8296.196,E2 -8296.196} C_VEL
LIN {X 0,Y 453.516,Z 129.616,A -85,B 0,C 180,E1 -8299.039,E2 -8299.039} C_VEL
LIN {X 0,Y 453.476,Z 129.62,A -85,B 0,C 180,E1 -8301.836,E2 -8301.836} C_VEL
LIN {X 0,Y 453.506,Z 129.623,A -85,B 0,C 180,E1 -8304.735,E2 -8304.735} C_VEL
LIN {X 0,Y 453.531,Z 129.614,A -85,B 0,C 180,E1 -8307.959,E2 -8307.959} C_VEL
LIN {X 0,Y 453.464,Z 129.621,A -85,B 0,C 180,E1 -8311.525,E2 -8311.525} C_VEL
LIN {X 0,Y 453.481,Z 129.621,A -85,B 0,C 180,E1 -8314.776,E2 -8314.776} C_VEL
LIN {X 0,Y 453.461,Z 129.616,A -85,B 0,C 180,E1 -8318.312,E2 -8318.312} C_VEL
LIN {X 0,Y 453.492,Z 129.624,A -85,B 0,C 180,E1 -8320.609,E2 -8320.609} C_VEL
LIN {X 0,Y 453.454,Z 129.615,A -85,B 0,C 180,E1 -8323.244,E2 -8323.244} C_VEL
LIN {X 0,Y 453.465,Z 129.625,A -85,B 0,C 180,E1 -8325.779,E2 -8325.779} C_VEL
LIN {X 0,Y 453.478,Z 129.625,A -85,B 0,C 180,E1 -8328.209,E2 -8328.209} C_VEL
LIN {X 0,Y 453.508,Z 129.62,A -85,B 0,C 180,E1 -8330.791,E2 -8330.791} C_VEL
LIN {X 0,Y 453.453,Z 129.63,A -85,B 0,C 180,E1 -8333.917,E2 -8333.917} C_VEL
LIN {X 0,Y 453.481,Z 129.619,A -85,B 0,C 180,E1 -8337.151,E2 -8337.151} C_VEL
LIN {X 0,Y 453.484,Z 129.706,A -85,B 0,C 180,E1 -8338.604,E2 -8338.604} C_VEL
LIN {X 0,Y 456.75,Z 142.16,A -85,B 0,C 180,E1 -8340.946,E2 -8340.946} C_VEL
LIN {X 0,Y 458.797,Z 151.948,A -85,B 0,C 180,E1 -8342.68,E2 -8342.68} C_VEL
LIN {X 0,Y 457.882,Z 166.385,A -85,B 0,C 180,E1 -8344.922,E2 -8344.922} C_VEL
LIN {X 0,Y 463.216,Z 193.21,A -85,B 0,C 180,E1 -8345.726,E2 -8345.726} C_VEL
LIN {X 0,Y 461.217,Z 333.442,A -85,B 0,C 180,E1 -8348.02,E2 -8348.02} C_VEL
LIN {X 0,Y 460.541,Z 349.225,A -85,B 0,C 180,E1 -8348.457,E2 -8348.457} C_VEL
LIN {X 0,Y 459.852,Z 364.069,A -85,B 0,C 180,E1 -8349.057,E2 -8349.057} C_VEL
LIN {X 0,Y 458.921,Z 378.861,A -85,B 0,C 180,E1 -8349.845,E2 -8349.845} C_VEL
LIN {X 0,Y 457.965,Z 392.128,A -85,B 0,C 180,E1 -8350.735,E2 -8350.735} C_VEL
LIN {X 0,Y 456.939,Z 405.655,A -85,B 0,C 180,E1 -8351.853,E2 -8351.853} C_VEL
LIN {X 0,Y 455.954,Z 417.978,A -85,B 0,C 180,E1 -8353.086,E2 -8353.086} C_VEL
LIN {X 0,Y 454.978,Z 430.067,A -85,B 0,C 180,E1 -8354.547,E2 -8354.547} C_VEL
LIN {X 0,Y 454.283,Z 439.441,A -85,B 0,C 180,E1 -8355.898,E2 -8355.898} C_VEL
LIN {X 0,Y 453.563,Z 448.654,A -85,B 0,C 180,E1 -8357.471,E2 -8357.471} C_VEL
LIN {X 0,Y 453.189,Z 457.344,A -85,B 0,C 180,E1 -8359.275,E2 -8359.275} C_VEL
LIN {X 0,Y 452.778,Z 464.321,A -85,B 0,C 180,E1 -8361.071,E2 -8361.071} C_VEL
LIN {X 0,Y 452.582,Z 469.813,A -85,B 0,C 180,E1 -8362.864,E2 -8362.864} C_VEL
LIN {X 0,Y 452.509,Z 473.972,A -85,B 0,C 180,E1 -8364.653,E2 -8364.653} C_VEL
LIN {X 0,Y 452.427,Z 476.883,A -85,B 0,C 180,E1 -8366.438,E2 -8366.438} C_VEL
LIN {X 0,Y 452.433,Z 478.617,A -85,B 0,C 180,E1 -8368.22,E2 -8368.22} C_VEL
LIN {X 0,Y 452.432,Z 479.205,A -85,B 0,C 180,E1 -8370,E2 -8370} C_VEL
LIN {X 0,Y 452.433,Z 478.595,A -85,B 0,C 180,E1 -8371.781,E2 -8371.781} C_VEL
LIN {X 0,Y 452.428,Z 476.824,A -85,B 0,C 180,E1 -8373.563,E2 -8373.563} C_VEL
LIN {X 0,Y 452.513,Z 473.872,A -85,B 0,C 180,E1 -8375.347,E2 -8375.347} C_VEL
LIN {X 0,Y 452.645,Z 469.667,A -85,B 0,C 180,E1 -8377.136,E2 -8377.136} C_VEL
LIN {X 0,Y 452.76,Z 464.091,A -85,B 0,C 180,E1 -8378.93,E2 -8378.93} C_VEL
LIN {X 0,Y 453.134,Z 457.002,A -85,B 0,C 180,E1 -8380.727,E2 -8380.727} C_VEL
LIN {X 0,Y 453.551,Z 449.12,A -85,B 0,C 180,E1 -8382.355,E2 -8382.355} C_VEL
LIN {X 0,Y 454.126,Z 440.252,A -85,B 0,C 180,E1 -8383.88,E2 -8383.88} C_VEL
LIN {X 0,Y 454.911,Z 429.193,A -85,B 0,C 180,E1 -8385.456,E2 -8385.456} C_VEL
LIN {X 0,Y 455.75,Z 417.824,A -85,B 0,C 180,E1 -8386.807,E2 -8386.807} C_VEL
LIN {X 0,Y 456.66,Z 405.325,A -85,B 0,C 180,E1 -8388.043,E2 -8388.043} C_VEL
LIN {X 0,Y 457.688,Z 391.494,A -85,B 0,C 180,E1 -8389.161,E2 -8389.161} C_VEL
LIN {X 0,Y 458.594,Z 377.903,A -85,B 0,C 180,E1 -8390.054,E2 -8390.054} C_VEL
LIN {X 0,Y 459.436,Z 363.957,A -85,B 0,C 180,E1 -8390.781,E2 -8390.781} C_VEL
LIN {X 0,Y 460.106,Z 348.483,A -85,B 0,C 180,E1 -8391.392,E2 -8391.392} C_VEL
LIN {X 0,Y 460.642,Z 333.268,A -85,B 0,C 180,E1 -8391.803,E2 -8391.803} C_VEL
LIN {X 0,Y 462.551,Z 193.668,A -85,B 0,C 180,E1 -8394.045,E2 -8394.045} C_VEL
LIN {X 0,Y 457.404,Z 166.729,A -85,B 0,C 180,E1 -8394.779,E2 -8394.779} C_VEL
LIN {X 0,Y 458.337,Z 150.663,A -85,B 0,C 180,E1 -8397.208,E2 -8397.208} C_VEL
LIN {X 0,Y 455.562,Z 138.196,A -85,B 0,C 180,E1 -8399.328,E2 -8399.328} C_VEL
LIN {X 0,Y 453.511,Z 129.62,A -85,B 0,C 180,E1 -8400.849,E2 -8400.849} C_VEL
LIN {X 0,Y 453.478,Z 129.627,A -85,B 0,C 180,E1 -8403.913,E2 -8403.913} C_VEL
LIN {X 0,Y 453.471,Z 129.626,A -85,B 0,C 180,E1 -8407.189,E2 -8407.189} C_VEL
LIN {X 0,Y 453.495,Z 129.619,A -85,B 0,C 180,E1 -8410.61,E2 -8410.61} C_VEL
LIN {X 0,Y 453.462,Z 129.626,A -85,B 0,C 180,E1 -8414.222,E2 -8414.222} C_VEL
LIN {X 0,Y 453.465,Z 129.626,A -85,B 0,C 180,E1 -8417.006,E2 -8417.006} C_VEL
LIN {X 0,Y 453.496,Z 129.624,A -85,B 0,C 180,E1 -8419.41,E2 -8419.41} C_VEL
LIN {X 0,Y 453.454,Z 129.623,A -85,B 0,C 180,E1 -8422.811,E2 -8422.811} C_VEL
LIN {X 0,Y 453.471,Z 129.621,A -85,B 0,C 180,E1 -8426.087,E2 -8426.087} C_VEL
LIN {X 0,Y 453.477,Z 129.624,A -85,B 0,C 180,E1 -8429.241,E2 -8429.241} C_VEL
LIN {X 0,Y 453.493,Z 129.605,A -85,B 0,C 180,E1 -8432.295,E2 -8432.295} C_VEL
LIN {X 0,Y 453.497,Z 129.62,A -85,B 0,C 180,E1 -8435.265,E2 -8435.265} C_VEL
LIN {X 0,Y 453.484,Z 129.617,A -85,B 0,C 180,E1 -8438.416,E2 -8438.416} C_VEL
LIN {X 0,Y 453.526,Z 129.617,A -85,B 0,C 180,E1 -8441.009,E2 -8441.009} C_VEL
LIN {X 0,Y 453.573,Z 129.605,A -85,B 0,C 180,E1 -8443.88,E2 -8443.88} C_VEL
LIN {X 0,Y 453.569,Z 129.605,A -85,B 0,C 180,E1 -8447.472,E2 -8447.472} C_VEL
LIN {X 0,Y 453.586,Z 129.605,A -85,B 0,C 180,E1 -8451.087,E2 -8451.087} C_VEL
LIN {X 0,Y 453.64,Z 129.599,A -85,B 0,C 180,E1 -8453.775,E2 -8453.775} C_VEL
LIN {X 0,Y 453.708,Z 129.585,A -85,B 0,C 180,E1 -8457.337,E2 -8457.337} C_VEL
LIN {X 0,Y 453.772,Z 129.569,A -85,B 0,C 180,E1 -8460,E2 -8460} C_VEL
LIN {X 0,Y 453.706,Z 129.59,A -85,B 0,C 180,E1 -8462.664,E2 -8462.664} C_VEL
LIN {X 0,Y 453.639,Z 129.598,A -85,B 0,C 180,E1 -8466.226,E2 -8466.226} C_VEL
LIN {X 0,Y 453.56,Z 129.593,A -85,B 0,C 180,E1 -8468.914,E2 -8468.914} C_VEL
LIN {X 0,Y 453.57,Z 129.605,A -85,B 0,C 180,E1 -8472.529,E2 -8472.529} C_VEL
LIN {X 0,Y 453.49,Z 129.616,A -85,B 0,C 180,E1 -8476.198,E2 -8476.198} C_VEL
LIN {X 0,Y 453.464,Z 129.621,A -85,B 0,C 180,E1 -8479.018,E2 -8479.018} C_VEL
LIN {X 0,Y 453.47,Z 129.62,A -85,B 0,C 180,E1 -8481.837,E2 -8481.837} C_VEL
LIN {X 0,Y 453.453,Z 129.623,A -85,B 0,C 180,E1 -8484.738,E2 -8484.738} C_VEL
LIN {X 0,Y 453.461,Z 129.612,A -85,B 0,C 180,E1 -8487.941,E2 -8487.941} C_VEL
LIN {X 0,Y 453.451,Z 129.612,A -85,B 0,C 180,E1 -8490.762,E2 -8490.762} C_VEL
LIN {X 0,Y 453.459,Z 129.622,A -85,B 0,C 180,E1 -8493.915,E2 -8493.915} C_VEL
LIN {X 0,Y 453.438,Z 129.616,A -85,B 0,C 180,E1 -8497.192,E2 -8497.192} C_VEL
LIN {X 0,Y 453.475,Z 129.618,A -85,B 0,C 180,E1 -8500.612,E2 -8500.612} C_VEL
LIN {X 0,Y 453.486,Z 129.62,A -85,B 0,C 180,E1 -8504.528,E2 -8504.528} C_VEL
LIN {X 0,Y 453.441,Z 129.623,A -85,B 0,C 180,E1 -8508.071,E2 -8508.071} C_VEL
LIN {X 0,Y 453.445,Z 129.623,A -85,B 0,C 180,E1 -8510.802,E2 -8510.802} C_VEL
LIN {X 0,Y 453.455,Z 129.621,A -85,B 0,C 180,E1 -8513.917,E2 -8513.917} C_VEL
LIN {X 0,Y 453.48,Z 129.613,A -85,B 0,C 180,E1 -8517.15,E2 -8517.15} C_VEL
LIN {X 0,Y 453.468,Z 129.628,A -85,B 0,C 180,E1 -8520.267,E2 -8520.267} C_VEL
LIN {X 0,Y 453.447,Z 129.626,A -85,B 0,C 180,E1 -8523.29,E2 -8523.29} C_VEL
LIN {X 0,Y 453.498,Z 129.624,A -85,B 0,C 180,E1 -8526.238,E2 -8526.238} C_VEL
LIN {X 0,Y 453.487,Z 129.619,A -85,B 0,C 180,E1 -8529.117,E2 -8529.117} C_VEL
LIN {X 0,Y 453.504,Z 129.611,A -85,B 0,C 180,E1 -8531.944,E2 -8531.944} C_VEL
LIN {X 0,Y 453.543,Z 129.613,A -85,B 0,C 180,E1 -8534.726,E2 -8534.726} C_VEL
LIN {X 0,Y 453.564,Z 129.613,A -85,B 0,C 180,E1 -8538.379,E2 -8538.379} C_VEL
LIN {X 0,Y 453.617,Z 129.755,A -85,B 0,C 180,E1 -8541.536,E2 -8541.536} C_VEL
LIN {X 0,Y 453.816,Z 130.602,A -85,B 0,C 180,E1 -8541.702,E2 -8541.702} C_VEL
LIN {X 0,Y 453.65,Z 132.924,A -85,B 0,C 180,E1 -8542.109,E2 -8542.109} C_VEL
LIN {X 0,Y 449.653,Z 141.268,A -85,B 0,C 180,E1 -8543.36,E2 -8543.36} C_VEL
LIN {X 0,Y 449.549,Z 143.601,A -85,B 0,C 180,E1 -8543.772,E2 -8543.772} C_VEL
LIN {X 0,Y 449.693,Z 144.228,A -85,B 0,C 180,E1 -8543.891,E2 -8543.891} C_VEL
LIN {X 0,Y 453.153,Z 154.05,A -85,B 0,C 180,E1 -8544.247,E2 -8544.247} C_VEL
LIN {X 0,Y 456.177,Z 167.294,A -85,B 0,C 180,E1 -8544.635,E2 -8544.635} C_VEL
LIN {X 0,Y 454.204,Z 309.163,A -85,B 0,C 180,E1 -8546.951,E2 -8546.951} C_VEL
LIN {X 0,Y 453.708,Z 324.188,A -85,B 0,C 180,E1 -8547.364,E2 -8547.364} C_VEL
LIN {X 0,Y 453.047,Z 339.995,A -85,B 0,C 180,E1 -8547.999,E2 -8547.999} C_VEL
LIN {X 0,Y 452.263,Z 354.444,A -85,B 0,C 180,E1 -8548.775,E2 -8548.775} C_VEL
LIN {X 0,Y 451.361,Z 367.64,A -85,B 0,C 180,E1 -8549.665,E2 -8549.665} C_VEL
LIN {X 0,Y 450.364,Z 381.113,A -85,B 0,C 180,E1 -8550.782,E2 -8550.782} C_VEL
LIN {X 0,Y 449.377,Z 393.335,A -85,B 0,C 180,E1 -8552.016,E2 -8552.016} C_VEL
LIN {X 0,Y 448.486,Z 404.481,A -85,B 0,C 180,E1 -8553.369,E2 -8553.369} C_VEL
LIN {X 0,Y 447.578,Z 415.391,A -85,B 0,C 180,E1 -8554.954,E2 -8554.954} C_VEL
LIN {X 0,Y 446.904,Z 424.437,A -85,B 0,C 180,E1 -8556.546,E2 -8556.546} C_VEL
LIN {X 0,Y 446.434,Z 431.97,A -85,B 0,C 180,E1 -8558.145,E2 -8558.145} C_VEL
LIN {X 0,Y 445.914,Z 439.07,A -85,B 0,C 180,E1 -8559.983,E2 -8559.983} C_VEL
LIN {X 0,Y 445.671,Z 444.653,A -85,B 0,C 180,E1 -8561.829,E2 -8561.829} C_VEL
LIN {X 0,Y 445.435,Z 448.888,A -85,B 0,C 180,E1 -8563.69,E2 -8563.69} C_VEL
LIN {X 0,Y 445.321,Z 452.007,A -85,B 0,C 180,E1 -8565.697,E2 -8565.697} C_VEL
LIN {X 0,Y 445.222,Z 453.56,A -85,B 0,C 180,E1 -8567.453,E2 -8567.453} C_VEL
LIN {X 0,Y 445.246,Z 454.039,A -85,B 0,C 180,E1 -8569.358,E2 -8569.358} C_VEL
LIN {X 0,Y 445.271,Z 453.179,A -85,B 0,C 180,E1 -8571.37,E2 -8571.37} C_VEL
LIN {X 0,Y 445.359,Z 451.139,A -85,B 0,C 180,E1 -8573.235,E2 -8573.235} C_VEL
LIN {X 0,Y 445.565,Z 447.602,A -85,B 0,C 180,E1 -8575.206,E2 -8575.206} C_VEL
LIN {X 0,Y 445.766,Z 443.909,A -85,B 0,C 180,E1 -8576.701,E2 -8576.701} C_VEL
LIN {X 0,Y 446.013,Z 439.312,A -85,B 0,C 180,E1 -8578.211,E2 -8578.211} C_VEL
LIN {X 0,Y 446.496,Z 432.397,A -85,B 0,C 180,E1 -8580.034,E2 -8580.034} C_VEL
LIN {X 0,Y 447.089,Z 425.182,A -85,B 0,C 180,E1 -8581.592,E2 -8581.592} C_VEL
LIN {X 0,Y 447.817,Z 415.528,A -85,B 0,C 180,E1 -8583.318,E2 -8583.318} C_VEL
LIN {X 0,Y 448.781,Z 405.055,A -85,B 0,C 180,E1 -8584.861,E2 -8584.861} C_VEL
LIN {X 0,Y 449.827,Z 393.489,A -85,B 0,C 180,E1 -8586.278,E2 -8586.278} C_VEL
LIN {X 0,Y 450.881,Z 380.677,A -85,B 0,C 180,E1 -8587.579,E2 -8587.579} C_VEL
LIN {X 0,Y 451.913,Z 367.819,A -85,B 0,C 180,E1 -8588.653,E2 -8588.653} C_VEL
LIN {X 0,Y 452.898,Z 354.12,A -85,B 0,C 180,E1 -8589.583,E2 -8589.583} C_VEL
LIN {X 0,Y 453.762,Z 339.603,A -85,B 0,C 180,E1 -8590.361,E2 -8590.361} C_VEL
LIN {X 0,Y 454.441,Z 324.191,A -85,B 0,C 180,E1 -8590.981,E2 -8590.981} C_VEL
LIN {X 0,Y 454.998,Z 308.987,A -85,B 0,C 180,E1 -8591.398,E2 -8591.398} C_VEL
LIN {X 0,Y 457.201,Z 167.745,A -85,B 0,C 180,E1 -8593.74,E2 -8593.74} C_VEL
LIN {X 0,Y 454.015,Z 154.267,A -85,B 0,C 180,E1 -8594.184,E2 -8594.184} C_VEL
LIN {X 0,Y 449.869,Z 144.639,A -85,B 0,C 180,E1 -8594.644,E2 -8594.644} C_VEL
LIN {X 0,Y 446.623,Z 131.379,A -85,B 0,C 180,E1 -8597.418,E2 -8597.418} C_VEL
LIN {X 0,Y 446.457,Z 130.502,A -85,B 0,C 180,E1 -8597.659,E2 -8597.659} C_VEL
LIN {X 0,Y 446.411,Z 130.509,A -85,B 0,C 180,E1 -8600.969,E2 -8600.969} C_VEL
LIN {X 0,Y 446.419,Z 130.501,A -85,B 0,C 180,E1 -8604.373,E2 -8604.373} C_VEL
LIN {X 0,Y 446.423,Z 130.498,A -85,B 0,C 180,E1 -8607.638,E2 -8607.638} C_VEL
LIN {X 0,Y 446.438,Z 130.495,A -85,B 0,C 180,E1 -8610.789,E2 -8610.789} C_VEL
LIN {X 0,Y 446.44,Z 130.502,A -85,B 0,C 180,E1 -8613.846,E2 -8613.846} C_VEL
LIN {X 0,Y 446.425,Z 130.495,A -85,B 0,C 180,E1 -8616.823,E2 -8616.823} C_VEL
LIN {X 0,Y 446.444,Z 130.498,A -85,B 0,C 180,E1 -8619.737,E2 -8619.737} C_VEL
LIN {X 0,Y 446.455,Z 130.494,A -85,B 0,C 180,E1 -8622.596,E2 -8622.596} C_VEL
LIN {X 0,Y 446.467,Z 130.493,A -85,B 0,C 180,E1 -8625.412,E2 -8625.412} C_VEL
LIN {X 0,Y 446.518,Z 130.487,A -85,B 0,C 180,E1 -8628.193,E2 -8628.193} C_VEL
LIN {X 0,Y 446.601,Z 130.48,A -85,B 0,C 180,E1 -8631.857,E2 -8631.857} C_VEL
LIN {X 0,Y 446.642,Z 130.467,A -85,B 0,C 180,E1 -8634.582,E2 -8634.582} C_VEL
LIN {X 0,Y 446.663,Z 130.466,A -85,B 0,C 180,E1 -8638.196,E2 -8638.196} C_VEL
LIN {X 0,Y 446.793,Z 130.454,A -85,B 0,C 180,E1 -8640,E2 -8640} C_VEL
LIN {X 0,Y 446.691,Z 130.465,A -85,B 0,C 180,E1 -8642.705,E2 -8642.705} C_VEL
LIN {X 0,Y 446.621,Z 130.473,A -85,B 0,C 180,E1 -8646.324,E2 -8646.324} C_VEL
LIN {X 0,Y 446.521,Z 130.486,A -85,B 0,C 180,E1 -8649.97,E2 -8649.97} C_VEL
LIN {X 0,Y 446.521,Z 130.486,A -85,B 0,C 180,E1 -8652.729,E2 -8652.729} C_VEL
LIN {X 0,Y 446.495,Z 130.486,A -85,B 0,C 180,E1 -8656.227,E2 -8656.227} C_VEL
LIN {X 0,Y 446.467,Z 130.491,A -85,B 0,C 180,E1 -8659.303,E2 -8659.303} C_VEL
LIN {X 0,Y 446.417,Z 130.5,A -85,B 0,C 180,E1 -8662.199,E2 -8662.199} C_VEL
LIN {X 0,Y 446.449,Z 130.497,A -85,B 0,C 180,E1 -8665.153,E2 -8665.153} C_VEL
LIN {X 0,Y 446.483,Z 130.494,A -85,B 0,C 180,E1 -8668.178,E2 -8668.178} C_VEL
LIN {X 0,Y 446.417,Z 130.499,A -85,B 0,C 180,E1 -8671.775,E2 -8671.775} C_VEL
LIN {X 0,Y 446.421,Z 130.502,A -85,B 0,C 180,E1 -8674.523,E2 -8674.523} C_VEL
LIN {X 0,Y 446.413,Z 130.495,A -85,B 0,C 180,E1 -8678.079,E2 -8678.079} C_VEL
LIN {X 0,Y 446.425,Z 130.502,A -85,B 0,C 180,E1 -8680.917,E2 -8680.917} C_VEL
LIN {X 0,Y 446.4,Z 130.496,A -85,B 0,C 180,E1 -8683.846,E2 -8683.846} C_VEL
LIN {X 0,Y 446.398,Z 130.499,A -85,B 0,C 180,E1 -8686.403,E2 -8686.403} C_VEL
LIN {X 0,Y 446.425,Z 130.499,A -85,B 0,C 180,E1 -8689.082,E2 -8689.082} C_VEL
LIN {X 0,Y 446.414,Z 130.504,A -85,B 0,C 180,E1 -8691.921,E2 -8691.921} C_VEL
LIN {X 0,Y 446.427,Z 130.498,A -85,B 0,C 180,E1 -8695.477,E2 -8695.477} C_VEL
LIN {X 0,Y 446.445,Z 130.594,A -85,B 0,C 180,E1 -8698.179,E2 -8698.179} C_VEL
LIN {X 0,Y 450.227,Z 145.008,A -85,B 0,C 180,E1 -8700.945,E2 -8700.945} C_VEL
LIN {X 0,Y 451.972,Z 153.109,A -85,B 0,C 180,E1 -8702.415,E2 -8702.415} C_VEL
LIN {X 0,Y 451.18,Z 166.202,A -85,B 0,C 180,E1 -8704.49,E2 -8704.49} C_VEL
LIN {X 0,Y 456.594,Z 192.894,A -85,B 0,C 180,E1 -8705.315,E2 -8705.315} C_VEL
LIN {X 0,Y 456.85,Z 198.251,A -85,B 0,C 180,E1 -8705.425,E2 -8705.425} C_VEL
LIN {X 0,Y 454.732,Z 333.138,A -85,B 0,C 180,E1 -8707.66,E2 -8707.66} C_VEL
LIN {X 0,Y 454.044,Z 348.95,A -85,B 0,C 180,E1 -8708.103,E2 -8708.103} C_VEL
LIN {X 0,Y 453.268,Z 363.599,A -85,B 0,C 180,E1 -8708.697,E2 -8708.697} C_VEL
LIN {X 0,Y 452.41,Z 377.215,A -85,B 0,C 180,E1 -8709.423,E2 -8709.423} C_VEL
LIN {X 0,Y 451.376,Z 390.715,A -85,B 0,C 180,E1 -8710.324,E2 -8710.324} C_VEL
LIN {X 0,Y 450.362,Z 403.176,A -85,B 0,C 180,E1 -8711.343,E2 -8711.343} C_VEL
LIN {X 0,Y 449.361,Z 414.79,A -85,B 0,C 180,E1 -8712.479,E2 -8712.479} C_VEL
LIN {X 0,Y 448.369,Z 426.496,A -85,B 0,C 180,E1 -8713.846,E2 -8713.846} C_VEL
LIN {X 0,Y 447.557,Z 436.371,A -85,B 0,C 180,E1 -8715.216,E2 -8715.216} C_VEL
LIN {X 0,Y 446.796,Z 446.072,A -85,B 0,C 180,E1 -8716.816,E2 -8716.816} C_VEL
LIN {X 0,Y 446.287,Z 454.176,A -85,B 0,C 180,E1 -8718.418,E2 -8718.418} C_VEL
LIN {X 0,Y 445.828,Z 460.9,A -85,B 0,C 180,E1 -8720.015,E2 -8720.015} C_VEL
LIN {X 0,Y 445.602,Z 467.098,A -85,B 0,C 180,E1 -8721.84,E2 -8721.84} C_VEL
LIN {X 0,Y 445.45,Z 471.996,A -85,B 0,C 180,E1 -8723.703,E2 -8723.703} C_VEL
LIN {X 0,Y 445.36,Z 475.403,A -85,B 0,C 180,E1 -8725.475,E2 -8725.475} C_VEL
LIN {X 0,Y 445.417,Z 477.71,A -85,B 0,C 180,E1 -8727.287,E2 -8727.287} C_VEL
LIN {X 0,Y 445.335,Z 478.857,A -85,B 0,C 180,E1 -8729.096,E2 -8729.096} C_VEL
LIN {X 0,Y 445.335,Z 478.848,A -85,B 0,C 180,E1 -8730.905,E2 -8730.905} C_VEL
LIN {X 0,Y 445.417,Z 477.645,A -85,B 0,C 180,E1 -8732.714,E2 -8732.714} C_VEL
LIN {X 0,Y 445.361,Z 475.275,A -85,B 0,C 180,E1 -8734.526,E2 -8734.526} C_VEL
LIN {X 0,Y 445.488,Z 471.694,A -85,B 0,C 180,E1 -8736.341,E2 -8736.341} C_VEL
LIN {X 0,Y 445.595,Z 466.8,A -85,B 0,C 180,E1 -8738.161,E2 -8738.161} C_VEL
LIN {X 0,Y 445.814,Z 460.463,A -85,B 0,C 180,E1 -8739.986,E2 -8739.986} C_VEL
LIN {X 0,Y 446.252,Z 453.635,A -85,B 0,C 180,E1 -8741.584,E2 -8741.584} C_VEL
LIN {X 0,Y 446.732,Z 445.355,A -85,B 0,C 180,E1 -8743.186,E2 -8743.186} C_VEL
LIN {X 0,Y 447.466,Z 435.411,A -85,B 0,C 180,E1 -8744.787,E2 -8744.787} C_VEL
LIN {X 0,Y 448.285,Z 425.219,A -85,B 0,C 180,E1 -8746.158,E2 -8746.158} C_VEL
LIN {X 0,Y 449.203,Z 413.317,A -85,B 0,C 180,E1 -8747.505,E2 -8747.505} C_VEL
LIN {X 0,Y 450.166,Z 400.963,A -85,B 0,C 180,E1 -8748.666,E2 -8748.666} C_VEL
LIN {X 0,Y 451.132,Z 387.79,A -85,B 0,C 180,E1 -8749.688,E2 -8749.688} C_VEL
LIN {X 0,Y 452.112,Z 373.29,A -85,B 0,C 180,E1 -8750.592,E2 -8750.592} C_VEL
LIN {X 0,Y 452.891,Z 359.384,A -85,B 0,C 180,E1 -8751.27,E2 -8751.27} C_VEL
LIN {X 0,Y 453.596,Z 343.885,A -85,B 0,C 180,E1 -8751.831,E2 -8751.831} C_VEL
LIN {X 0,Y 454.094,Z 328.721,A -85,B 0,C 180,E1 -8752.194,E2 -8752.194} C_VEL
LIN {X 0,Y 455.953,Z 195.246,A -85,B 0,C 180,E1 -8754.356,E2 -8754.356} C_VEL
LIN {X 0,Y 453.384,Z 181,A -85,B 0,C 180,E1 -8754.733,E2 -8754.733} C_VEL
LIN {X 0,Y 450.663,Z 166.597,A -85,B 0,C 180,E1 -8755.135,E2 -8755.135} C_VEL
LIN {X 0,Y 451.517,Z 152.661,A -85,B 0,C 180,E1 -8757.275,E2 -8757.275} C_VEL
LIN {X 0,Y 448.987,Z 140.951,A -85,B 0,C 180,E1 -8759.286,E2 -8759.286} C_VEL
LIN {X 0,Y 446.454,Z 130.498,A -85,B 0,C 180,E1 -8761.166,E2 -8761.166} C_VEL
LIN {X 0,Y 446.431,Z 130.505,A -85,B 0,C 180,E1 -8764.523,E2 -8764.523} C_VEL
LIN {X 0,Y 446.429,Z 130.501,A -85,B 0,C 180,E1 -8768.082,E2 -8768.082} C_VEL
LIN {X 0,Y 446.424,Z 130.5,A -85,B 0,C 180,E1 -8770.917,E2 -8770.917} C_VEL
LIN {X 0,Y 446.401,Z 130.508,A -85,B 0,C 180,E1 -8773.847,E2 -8773.847} C_VEL
LIN {X 0,Y 446.4,Z 130.504,A -85,B 0,C 180,E1 -8776.404,E2 -8776.404} C_VEL
LIN {X 0,Y 446.429,Z 130.503,A -85,B 0,C 180,E1 -8779.083,E2 -8779.083} C_VEL
LIN {X 0,Y 446.41,Z 130.5,A -85,B 0,C 180,E1 -8782.122,E2 -8782.122} C_VEL
LIN {X 0,Y 446.426,Z 130.503,A -85,B 0,C 180,E1 -8785.477,E2 -8785.477} C_VEL
LIN {X 0,Y 446.417,Z 130.5,A -85,B 0,C 180,E1 -8788.7,E2 -8788.7} C_VEL
LIN {X 0,Y 446.45,Z 130.482,A -85,B 0,C 180,E1 -8791.831,E2 -8791.831} C_VEL
LIN {X 0,Y 446.442,Z 130.496,A -85,B 0,C 180,E1 -8794.847,E2 -8794.847} C_VEL
LIN {X 0,Y 446.452,Z 130.492,A -85,B 0,C 180,E1 -8798.246,E2 -8798.246} C_VEL
LIN {X 0,Y 446.453,Z 130.493,A -85,B 0,C 180,E1 -8801.649,E2 -8801.649} C_VEL
LIN {X 0,Y 446.509,Z 130.489,A -85,B 0,C 180,E1 -8804.48,E2 -8804.48} C_VEL
LIN {X 0,Y 446.521,Z 130.485,A -85,B 0,C 180,E1 -8808.193,E2 -8808.193} C_VEL
LIN {X 0,Y 446.534,Z 130.485,A -85,B 0,C 180,E1 -8810.945,E2 -8810.945} C_VEL
LIN {X 0,Y 446.61,Z 130.474,A -85,B 0,C 180,E1 -8813.676,E2 -8813.676} C_VEL
LIN {X 0,Y 446.657,Z 130.463,A -85,B 0,C 180,E1 -8817.295,E2 -8817.295} C_VEL
LIN {X 0,Y 446.722,Z 130.446,A -85,B 0,C 180,E1 -8820,E2 -8820} C_VEL
LIN {X 0,Y 446.655,Z 130.468,A -85,B 0,C 180,E1 -8822.706,E2 -8822.706} C_VEL
LIN {X 0,Y 446.609,Z 130.473,A -85,B 0,C 180,E1 -8826.325,E2 -8826.325} C_VEL
LIN {X 0,Y 446.511,Z 130.471,A -85,B 0,C 180,E1 -8829.056,E2 -8829.056} C_VEL
LIN {X 0,Y 446.497,Z 130.486,A -85,B 0,C 180,E1 -8832.731,E2 -8832.731} C_VEL
LIN {X 0,Y 446.459,Z 130.491,A -85,B 0,C 180,E1 -8836.209,E2 -8836.209} C_VEL
LIN {X 0,Y 446.405,Z 130.503,A -85,B 0,C 180,E1 -8839.307,E2 -8839.307} C_VEL
LIN {X 0,Y 446.407,Z 130.497,A -85,B 0,C 180,E1 -8842.201,E2 -8842.201} C_VEL
LIN {X 0,Y 446.41,Z 130.504,A -85,B 0,C 180,E1 -8845.156,E2 -8845.156} C_VEL
LIN {X 0,Y 446.42,Z 130.487,A -85,B 0,C 180,E1 -8848.184,E2 -8848.184} C_VEL
LIN {X 0,Y 446.393,Z 130.498,A -85,B 0,C 180,E1 -8851.303,E2 -8851.303} C_VEL
LIN {X 0,Y 446.417,Z 130.5,A -85,B 0,C 180,E1 -8854.525,E2 -8854.525} C_VEL
LIN {X 0,Y 446.401,Z 130.486,A -85,B 0,C 180,E1 -8858.076,E2 -8858.076} C_VEL
LIN {X 0,Y 446.405,Z 130.502,A -85,B 0,C 180,E1 -8861.394,E2 -8861.394} C_VEL
LIN {X 0,Y 446.426,Z 130.489,A -85,B 0,C 180,E1 -8865.108,E2 -8865.108} C_VEL
LIN {X 0,Y 446.405,Z 130.505,A -85,B 0,C 180,E1 -8868.606,E2 -8868.606} C_VEL
LIN {X 0,Y 446.41,Z 130.495,A -85,B 0,C 180,E1 -8871.923,E2 -8871.923} C_VEL
LIN {X 0,Y 446.427,Z 130.498,A -85,B 0,C 180,E1 -8875.476,E2 -8875.476} C_VEL
LIN {X 0,Y 446.42,Z 130.504,A -85,B 0,C 180,E1 -8878.699,E2 -8878.699} C_VEL
LIN {X 0,Y 446.429,Z 130.498,A -85,B 0,C 180,E1 -8881.836,E2 -8881.836} C_VEL
LIN {X 0,Y 446.427,Z 130.501,A -85,B 0,C 180,E1 -8884.845,E2 -8884.845} C_VEL
LIN {X 0,Y 446.454,Z 130.5,A -85,B 0,C 180,E1 -8888.245,E2 -8888.245} C_VEL
LIN {X 0,Y 446.454,Z 130.491,A -85,B 0,C 180,E1 -8891.649,E2 -8891.649} C_VEL
LIN {X 0,Y 446.512,Z 130.49,A -85,B 0,C 180,E1 -8894.479,E2 -8894.479} C_VEL
LIN {X 0,Y 446.523,Z 130.49,A -85,B 0,C 180,E1 -8898.193,E2 -8898.193} C_VEL
LIN {X 0,Y 446.573,Z 130.607,A -85,B 0,C 180,E1 -8901.23,E2 -8901.23} C_VEL
LIN {X 0,Y 449.549,Z 143.601,A -85,B 0,C 180,E1 -8903.772,E2 -8903.772} C_VEL
LIN {X 0,Y 450.628,Z 145.229,A -85,B 0,C 180,E1 -8903.958,E2 -8903.958} C_VEL
LIN {X 0,Y 453.826,Z 149.633,A -85,B 0,C 180,E1 -8904.208,E2 -8904.208} C_VEL
LIN {X 0,Y 455.398,Z 153.395,A -85,B 0,C 180,E1 -8904.356,E2 -8904.356} C_VEL
LIN {X 0,Y 455.813,Z 157.667,A -85,B 0,C 180,E1 -8904.449,E2 -8904.449} C_VEL
LIN {X 0,Y 454.772,Z 162.048,A -85,B 0,C 180,E1 -8904.43,E2 -8904.43} C_VEL
LIN {X 0,Y 450.19,Z 171.627,A -85,B 0,C 180,E1 -8904.38,E2 -8904.38} C_VEL
LIN {X 0,Y 449.525,Z 175.033,A -85,B 0,C 180,E1 -8904.412,E2 -8904.412} C_VEL
LIN {X 0,Y 447.543,Z 309.986,A -85,B 0,C 180,E1 -8906.652,E2 -8906.652} C_VEL
LIN {X 0,Y 447.046,Z 324.808,A -85,B 0,C 180,E1 -8907.071,E2 -8907.071} C_VEL
LIN {X 0,Y 446.357,Z 339.927,A -85,B 0,C 180,E1 -8907.687,E2 -8907.687} C_VEL
LIN {X 0,Y 445.6,Z 353.472,A -85,B 0,C 180,E1 -8908.418,E2 -8908.418} C_VEL
LIN {X 0,Y 444.649,Z 366.881,A -85,B 0,C 180,E1 -8909.32,E2 -8909.32} C_VEL
LIN {X 0,Y 443.592,Z 380.536,A -85,B 0,C 180,E1 -8910.454,E2 -8910.454} C_VEL
LIN {X 0,Y 442.592,Z 392.758,A -85,B 0,C 180,E1 -8911.691,E2 -8911.691} C_VEL
LIN {X 0,Y 441.689,Z 403.284,A -85,B 0,C 180,E1 -8912.964,E2 -8912.964} C_VEL
LIN {X 0,Y 440.852,Z 412.955,A -85,B 0,C 180,E1 -8914.342,E2 -8914.342} C_VEL
LIN {X 0,Y 440.139,Z 422.444,A -85,B 0,C 180,E1 -8915.957,E2 -8915.957} C_VEL
LIN {X 0,Y 439.532,Z 430.17,A -85,B 0,C 180,E1 -8917.531,E2 -8917.531} C_VEL
LIN {X 0,Y 439.009,Z 437.014,A -85,B 0,C 180,E1 -8919.212,E2 -8919.212} C_VEL
LIN {X 0,Y 438.698,Z 443.104,A -85,B 0,C 180,E1 -8921.083,E2 -8921.083} C_VEL
LIN {X 0,Y 438.457,Z 447.797,A -85,B 0,C 180,E1 -8922.968,E2 -8922.968} C_VEL
LIN {X 0,Y 438.276,Z 451.177,A -85,B 0,C 180,E1 -8924.866,E2 -8924.866} C_VEL
LIN {X 0,Y 438.164,Z 453.31,A -85,B 0,C 180,E1 -8926.781,E2 -8926.781} C_VEL
LIN {X 0,Y 438.183,Z 454.234,A -85,B 0,C 180,E1 -8928.861,E2 -8928.861} C_VEL
LIN {X 0,Y 438.152,Z 453.853,A -85,B 0,C 180,E1 -8930.663,E2 -8930.663} C_VEL
LIN {X 0,Y 438.235,Z 452.198,A -85,B 0,C 180,E1 -8932.637,E2 -8932.637} C_VEL
LIN {X 0,Y 438.391,Z 449.16,A -85,B 0,C 180,E1 -8934.633,E2 -8934.633} C_VEL
LIN {X 0,Y 438.678,Z 444.622,A -85,B 0,C 180,E1 -8936.653,E2 -8936.653} C_VEL
LIN {X 0,Y 439.059,Z 438.421,A -85,B 0,C 180,E1 -8938.699,E2 -8938.699} C_VEL
LIN {X 0,Y 439.569,Z 431.537,A -85,B 0,C 180,E1 -8940.483,E2 -8940.483} C_VEL
LIN {X 0,Y 440.262,Z 423.342,A -85,B 0,C 180,E1 -8942.214,E2 -8942.214} C_VEL
LIN {X 0,Y 441.185,Z 413.731,A -85,B 0,C 180,E1 -8943.886,E2 -8943.886} C_VEL
LIN {X 0,Y 442.139,Z 402.809,A -85,B 0,C 180,E1 -8945.463,E2 -8945.463} C_VEL
LIN {X 0,Y 443.186,Z 391.923,A -85,B 0,C 180,E1 -8946.772,E2 -8946.772} C_VEL
LIN {X 0,Y 444.21,Z 380.229,A -85,B 0,C 180,E1 -8947.956,E2 -8947.956} C_VEL
LIN {X 0,Y 445.3,Z 367.807,A -85,B 0,C 180,E1 -8949.001,E2 -8949.001} C_VEL
LIN {X 0,Y 446.333,Z 354.253,A -85,B 0,C 180,E1 -8949.933,E2 -8949.933} C_VEL
LIN {X 0,Y 447.233,Z 340.212,A -85,B 0,C 180,E1 -8950.699,E2 -8950.699} C_VEL
LIN {X 0,Y 447.939,Z 324.875,A -85,B 0,C 180,E1 -8951.333,E2 -8951.333} C_VEL
LIN {X 0,Y 448.541,Z 309.212,A -85,B 0,C 180,E1 -8951.771,E2 -8951.771} C_VEL
LIN {X 0,Y 450.855,Z 168.988,A -85,B 0,C 180,E1 -8954.13,E2 -8954.13} C_VEL
LIN {X 0,Y 448.13,Z 157.187,A -85,B 0,C 180,E1 -8954.528,E2 -8954.528} C_VEL
LIN {X 0,Y 442.741,Z 144.882,A -85,B 0,C 180,E1 -8955.138,E2 -8955.138} C_VEL
LIN {X 0,Y 439.396,Z 131.429,A -85,B 0,C 180,E1 -8958.021,E2 -8958.021} C_VEL
LIN {X 0,Y 439.364,Z 131.386,A -85,B 0,C 180,E1 -8961.402,E2 -8961.402} C_VEL
LIN {X 0,Y 439.399,Z 131.37,A -85,B 0,C 180,E1 -8964.843,E2 -8964.843} C_VEL
LIN {X 0,Y 439.374,Z 131.374,A -85,B 0,C 180,E1 -8968.139,E2 -8968.139} C_VEL
LIN {X 0,Y 439.41,Z 131.367,A -85,B 0,C 180,E1 -8971.603,E2 -8971.603} C_VEL
LIN {X 0,Y 439.378,Z 131.377,A -85,B 0,C 180,E1 -8974.413,E2 -8974.413} C_VEL
LIN {X 0,Y 439.364,Z 131.376,A -85,B 0,C 180,E1 -8977.424,E2 -8977.424} C_VEL
LIN {X 0,Y 439.441,Z 131.37,A -85,B 0,C 180,E1 -8980.663,E2 -8980.663} C_VEL
LIN {X 0,Y 439.462,Z 131.366,A -85,B 0,C 180,E1 -8984.224,E2 -8984.224} C_VEL
LIN {X 0,Y 439.484,Z 131.363,A -85,B 0,C 180,E1 -8988.001,E2 -8988.001} C_VEL
LIN {X 0,Y 439.548,Z 131.357,A -85,B 0,C 180,E1 -8991.726,E2 -8991.726} C_VEL
LIN {X 0,Y 439.617,Z 131.342,A -85,B 0,C 180,E1 -8994.495,E2 -8994.495} C_VEL
LIN {X 0,Y 439.633,Z 131.342,A -85,B 0,C 180,E1 -8998.167,E2 -8998.167} C_VEL
LIN {X 0,Y 439.763,Z 131.329,A -85,B 0,C 180,E1 -9000,E2 -9000} C_VEL
LIN {X 0,Y 439.64,Z 131.343,A -85,B 0,C 180,E1 -9002.748,E2 -9002.748} C_VEL
LIN {X 0,Y 439.593,Z 131.349,A -85,B 0,C 180,E1 -9006.425,E2 -9006.425} C_VEL
LIN {X 0,Y 439.495,Z 131.362,A -85,B 0,C 180,E1 -9009.201,E2 -9009.201} C_VEL
LIN {X 0,Y 439.465,Z 131.365,A -85,B 0,C 180,E1 -9012.937,E2 -9012.937} C_VEL
LIN {X 0,Y 439.446,Z 131.364,A -85,B 0,C 180,E1 -9016.348,E2 -9016.348} C_VEL
LIN {X 0,Y 439.401,Z 131.37,A -85,B 0,C 180,E1 -9019.626,E2 -9019.626} C_VEL
LIN {X 0,Y 439.364,Z 131.38,A -85,B 0,C 180,E1 -9022.575,E2 -9022.575} C_VEL
LIN {X 0,Y 439.399,Z 131.372,A -85,B 0,C 180,E1 -9025.585,E2 -9025.585} C_VEL
LIN {X 0,Y 439.416,Z 131.374,A -85,B 0,C 180,E1 -9028.673,E2 -9028.673} C_VEL
LIN {X 0,Y 439.367,Z 131.378,A -85,B 0,C 180,E1 -9032.03,E2 -9032.03} C_VEL
LIN {X 0,Y 439.39,Z 131.375,A -85,B 0,C 180,E1 -9035.34,E2 -9035.34} C_VEL
LIN {X 0,Y 439.375,Z 131.368,A -85,B 0,C 180,E1 -9038.595,E2 -9038.595} C_VEL
LIN {X 0,Y 439.387,Z 131.377,A -85,B 0,C 180,E1 -9041.257,E2 -9041.257} C_VEL
LIN {X 0,Y 439.4,Z 131.378,A -85,B 0,C 180,E1 -9044.729,E2 -9044.729} C_VEL
LIN {X 0,Y 439.394,Z 131.374,A -85,B 0,C 180,E1 -9047.796,E2 -9047.796} C_VEL
LIN {X 0,Y 439.428,Z 131.369,A -85,B 0,C 180,E1 -9050.228,E2 -9050.228} C_VEL
LIN {X 0,Y 439.372,Z 131.381,A -85,B 0,C 180,E1 -9053.713,E2 -9053.713} C_VEL
LIN {X 0,Y 439.371,Z 131.377,A -85,B 0,C 180,E1 -9057.054,E2 -9057.054} C_VEL
LIN {X 0,Y 439.393,Z 131.524,A -85,B 0,C 180,E1 -9057.742,E2 -9057.742} C_VEL
LIN {X 0,Y 442.825,Z 144.281,A -85,B 0,C 180,E1 -9060.267,E2 -9060.267} C_VEL
LIN {X 0,Y 445.25,Z 155.585,A -85,B 0,C 180,E1 -9062.361,E2 -9062.361} C_VEL
LIN {X 0,Y 444.535,Z 166.151,A -85,B 0,C 180,E1 -9064.041,E2 -9064.041} C_VEL
LIN {X 0,Y 449.336,Z 189.117,A -85,B 0,C 180,E1 -9064.784,E2 -9064.784} C_VEL
LIN {X 0,Y 450.525,Z 195.724,A -85,B 0,C 180,E1 -9064.979,E2 -9064.979} C_VEL
LIN {X 0,Y 448.275,Z 332.977,A -85,B 0,C 180,E1 -9067.29,E2 -9067.29} C_VEL
LIN {X 0,Y 447.525,Z 348.747,A -85,B 0,C 180,E1 -9067.737,E2 -9067.737} C_VEL
LIN {X 0,Y 446.648,Z 364.233,A -85,B 0,C 180,E1 -9068.382,E2 -9068.382} C_VEL
LIN {X 0,Y 445.782,Z 377.455,A -85,B 0,C 180,E1 -9069.103,E2 -9069.103} C_VEL
LIN {X 0,Y 444.673,Z 390.868,A -85,B 0,C 180,E1 -9070.015,E2 -9070.015} C_VEL
LIN {X 0,Y 443.497,Z 404.553,A -85,B 0,C 180,E1 -9071.163,E2 -9071.163} C_VEL
LIN {X 0,Y 442.353,Z 416.963,A -85,B 0,C 180,E1 -9072.431,E2 -9072.431} C_VEL
LIN {X 0,Y 441.353,Z 428.28,A -85,B 0,C 180,E1 -9073.82,E2 -9073.82} C_VEL
LIN {X 0,Y 440.394,Z 439.313,A -85,B 0,C 180,E1 -9075.443,E2 -9075.443} C_VEL
LIN {X 0,Y 439.601,Z 448.465,A -85,B 0,C 180,E1 -9077.067,E2 -9077.067} C_VEL
LIN {X 0,Y 439.105,Z 457.104,A -85,B 0,C 180,E1 -9078.927,E2 -9078.927} C_VEL
LIN {X 0,Y 438.634,Z 464.048,A -85,B 0,C 180,E1 -9080.78,E2 -9080.78} C_VEL
LIN {X 0,Y 438.427,Z 469.512,A -85,B 0,C 180,E1 -9082.632,E2 -9082.632} C_VEL
LIN {X 0,Y 438.312,Z 473.64,A -85,B 0,C 180,E1 -9084.48,E2 -9084.48} C_VEL
LIN {X 0,Y 438.229,Z 476.525,A -85,B 0,C 180,E1 -9086.322,E2 -9086.322} C_VEL
LIN {X 0,Y 438.274,Z 478.236,A -85,B 0,C 180,E1 -9088.162,E2 -9088.162} C_VEL
LIN {X 0,Y 438.25,Z 478.803,A -85,B 0,C 180,E1 -9090,E2 -9090} C_VEL
LIN {X 0,Y 438.274,Z 478.18,A -85,B 0,C 180,E1 -9091.838,E2 -9091.838} C_VEL
LIN {X 0,Y 438.231,Z 476.382,A -85,B 0,C 180,E1 -9093.678,E2 -9093.678} C_VEL
LIN {X 0,Y 438.321,Z 473.401,A -85,B 0,C 180,E1 -9095.521,E2 -9095.521} C_VEL
LIN {X 0,Y 438.482,Z 469.162,A -85,B 0,C 180,E1 -9097.367,E2 -9097.367} C_VEL
LIN {X 0,Y 438.622,Z 463.546,A -85,B 0,C 180,E1 -9099.221,E2 -9099.221} C_VEL
LIN {X 0,Y 439.082,Z 456.411,A -85,B 0,C 180,E1 -9101.074,E2 -9101.074} C_VEL
LIN {X 0,Y 439.478,Z 448.721,A -85,B 0,C 180,E1 -9102.712,E2 -9102.712} C_VEL
LIN {X 0,Y 440.196,Z 439.571,A -85,B 0,C 180,E1 -9104.328,E2 -9104.328} C_VEL
LIN {X 0,Y 440.899,Z 430.156,A -85,B 0,C 180,E1 -9105.723,E2 -9105.723} C_VEL
LIN {X 0,Y 441.872,Z 418.496,A -85,B 0,C 180,E1 -9107.175,E2 -9107.175} C_VEL
LIN {X 0,Y 442.907,Z 405.626,A -85,B 0,C 180,E1 -9108.504,E2 -9108.504} C_VEL
LIN {X 0,Y 444.051,Z 391.956,A -85,B 0,C 180,E1 -9109.654,E2 -9109.654} C_VEL
LIN {X 0,Y 445.03,Z 378.508,A -85,B 0,C 180,E1 -9110.572,E2 -9110.572} C_VEL
LIN {X 0,Y 445.949,Z 364.279,A -85,B 0,C 180,E1 -9111.344,E2 -9111.344} C_VEL
LIN {X 0,Y 446.715,Z 348.419,A -85,B 0,C 180,E1 -9111.995,E2 -9111.995} C_VEL
LIN {X 0,Y 447.322,Z 332.904,A -85,B 0,C 180,E1 -9112.426,E2 -9112.426} C_VEL
LIN {X 0,Y 449.392,Z 196.194,A -85,B 0,C 180,E1 -9114.684,E2 -9114.684} C_VEL
LIN {X 0,Y 445.106,Z 173.068,A -85,B 0,C 180,E1 -9115.318,E2 -9115.318} C_VEL
LIN {X 0,Y 443.895,Z 166.369,A -85,B 0,C 180,E1 -9115.517,E2 -9115.517} C_VEL
LIN {X 0,Y 444.615,Z 153.681,A -85,B 0,C 180,E1 -9117.497,E2 -9117.497} C_VEL
LIN {X 0,Y 441.63,Z 140.559,A -85,B 0,C 180,E1 -9119.807,E2 -9119.807} C_VEL
LIN {X 0,Y 439.397,Z 131.378,A -85,B 0,C 180,E1 -9121.489,E2 -9121.489} C_VEL
LIN {X 0,Y 439.389,Z 131.382,A -85,B 0,C 180,E1 -9124.044,E2 -9124.044} C_VEL
LIN {X 0,Y 439.361,Z 131.386,A -85,B 0,C 180,E1 -9127.435,E2 -9127.435} C_VEL
LIN {X 0,Y 439.403,Z 131.379,A -85,B 0,C 180,E1 -9129.85,E2 -9129.85} C_VEL
LIN {X 0,Y 439.372,Z 131.378,A -85,B 0,C 180,E1 -9132.626,E2 -9132.626} C_VEL
LIN {X 0,Y 439.401,Z 131.38,A -85,B 0,C 180,E1 -9135.271,E2 -9135.271} C_VEL
LIN {X 0,Y 439.391,Z 131.377,A -85,B 0,C 180,E1 -9138.744,E2 -9138.744} C_VEL
LIN {X 0,Y 439.371,Z 131.378,A -85,B 0,C 180,E1 -9141.609,E2 -9141.609} C_VEL
LIN {X 0,Y 439.399,Z 131.374,A -85,B 0,C 180,E1 -9144.844,E2 -9144.844} C_VEL
LIN {X 0,Y 439.374,Z 131.376,A -85,B 0,C 180,E1 -9148.14,E2 -9148.14} C_VEL
LIN {X 0,Y 439.403,Z 131.361,A -85,B 0,C 180,E1 -9151.606,E2 -9151.606} C_VEL
LIN {X 0,Y 439.38,Z 131.371,A -85,B 0,C 180,E1 -9154.414,E2 -9154.414} C_VEL
LIN {X 0,Y 439.367,Z 131.375,A -85,B 0,C 180,E1 -9157.425,E2 -9157.425} C_VEL
LIN {X 0,Y 439.445,Z 131.372,A -85,B 0,C 180,E1 -9160.664,E2 -9160.664} C_VEL
LIN {X 0,Y 439.465,Z 131.364,A -85,B 0,C 180,E1 -9164.225,E2 -9164.225} C_VEL
LIN {X 0,Y 439.488,Z 131.36,A -85,B 0,C 180,E1 -9168.002,E2 -9168.002} C_VEL
LIN {X 0,Y 439.507,Z 131.358,A -85,B 0,C 180,E1 -9171.726,E2 -9171.726} C_VEL
LIN {X 0,Y 439.6,Z 131.354,A -85,B 0,C 180,E1 -9174.496,E2 -9174.496} C_VEL
LIN {X 0,Y 439.631,Z 131.335,A -85,B 0,C 180,E1 -9178.168,E2 -9178.168} C_VEL
LIN {X 0,Y 439.673,Z 131.323,A -85,B 0,C 180,E1 -9180,E2 -9180} C_VEL
LIN {X 0,Y 439.607,Z 131.346,A -85,B 0,C 180,E1 -9182.749,E2 -9182.749} C_VEL
LIN {X 0,Y 439.563,Z 131.349,A -85,B 0,C 180,E1 -9186.426,E2 -9186.426} C_VEL
LIN {X 0,Y 439.477,Z 131.347,A -85,B 0,C 180,E1 -9189.203,E2 -9189.203} C_VEL
LIN {X 0,Y 439.456,Z 131.363,A -85,B 0,C 180,E1 -9192.938,E2 -9192.938} C_VEL
LIN {X 0,Y 439.4,Z 131.37,A -85,B 0,C 180,E1 -9196.325,E2 -9196.325} C_VEL
LIN {X 0,Y 439.36,Z 131.384,A -85,B 0,C 180,E1 -9199.629,E2 -9199.629} C_VEL
LIN {X 0,Y 439.352,Z 131.375,A -85,B 0,C 180,E1 -9202.577,E2 -9202.577} C_VEL
LIN {X 0,Y 439.354,Z 131.381,A -85,B 0,C 180,E1 -9205.589,E2 -9205.589} C_VEL
LIN {X 0,Y 439.381,Z 131.365,A -85,B 0,C 180,E1 -9208.677,E2 -9208.677} C_VEL
LIN {X 0,Y 439.347,Z 131.376,A -85,B 0,C 180,E1 -9212.024,E2 -9212.024} C_VEL
LIN {X 0,Y 439.388,Z 131.375,A -85,B 0,C 180,E1 -9215.338,E2 -9215.338} C_VEL
LIN {X 0,Y 439.358,Z 131.365,A -85,B 0,C 180,E1 -9218.598,E2 -9218.598} C_VEL
LIN {X 0,Y 439.354,Z 131.379,A -85,B 0,C 180,E1 -9222.21,E2 -9222.21} C_VEL
LIN {X 0,Y 439.38,Z 131.365,A -85,B 0,C 180,E1 -9225.267,E2 -9225.267} C_VEL
LIN {X 0,Y 439.368,Z 131.384,A -85,B 0,C 180,E1 -9228.747,E2 -9228.747} C_VEL
LIN {X 0,Y 439.365,Z 131.372,A -85,B 0,C 180,E1 -9231.61,E2 -9231.61} C_VEL
LIN {X 0,Y 439.4,Z 131.376,A -85,B 0,C 180,E1 -9234.844,E2 -9234.844} C_VEL
LIN {X 0,Y 439.375,Z 131.374,A -85,B 0,C 180,E1 -9238.139,E2 -9238.139} C_VEL
LIN {X 0,Y 439.405,Z 131.372,A -85,B 0,C 180,E1 -9241.606,E2 -9241.606} C_VEL
LIN {X 0,Y 439.372,Z 131.383,A -85,B 0,C 180,E1 -9244.413,E2 -9244.413} C_VEL
LIN {X 0,Y 439.369,Z 131.38,A -85,B 0,C 180,E1 -9247.424,E2 -9247.424} C_VEL
LIN {X 0,Y 439.446,Z 131.367,A -85,B 0,C 180,E1 -9250.663,E2 -9250.663} C_VEL
LIN {X 0,Y 439.467,Z 131.37,A -85,B 0,C 180,E1 -9254.224,E2 -9254.224} C_VEL
LIN {X 0,Y 439.489,Z 131.368,A -85,B 0,C 180,E1 -9258.001,E2 -9258.001} C_VEL
LIN {X 0,Y 439.518,Z 131.446,A -85,B 0,C 180,E1 -9260.914,E2 -9260.914} C_VEL
LIN {X 0,Y 442.457,Z 144.368,A -85,B 0,C 180,E1 -9263.48,E2 -9263.48} C_VEL
LIN {X 0,Y 446.808,Z 156.024,A -85,B 0,C 180,E1 -9263.935,E2 -9263.935} C_VEL
LIN {X 0,Y 449.642,Z 168.708,A -85,B 0,C 180,E1 -9264.309,E2 -9264.309} C_VEL
LIN {X 0,Y 449.525,Z 175.033,A -85,B 0,C 180,E1 -9264.412,E2 -9264.412} C_VEL
LIN {X 0,Y 448.723,Z 180.889,A -85,B 0,C 180,E1 -9264.469,E2 -9264.469} C_VEL
LIN {X 0,Y 443.106,Z 199.929,A -85,B 0,C 180,E1 -9264.498,E2 -9264.498} C_VEL
LIN {X 0,Y 442.538,Z 205.77,A -85,B 0,C 180,E1 -9264.569,E2 -9264.569} C_VEL
LIN {X 0,Y 440.938,Z 309.612,A -85,B 0,C 180,E1 -9266.316,E2 -9266.316} C_VEL
LIN {X 0,Y 440.39,Z 324.629,A -85,B 0,C 180,E1 -9266.74,E2 -9266.74} C_VEL
LIN {X 0,Y 439.686,Z 339.844,A -85,B 0,C 180,E1 -9267.366,E2 -9267.366} C_VEL
LIN {X 0,Y 438.837,Z 354.409,A -85,B 0,C 180,E1 -9268.164,E2 -9268.164} C_VEL
LIN {X 0,Y 437.84,Z 367.682,A -85,B 0,C 180,E1 -9269.08,E2 -9269.08} C_VEL
LIN {X 0,Y 436.739,Z 381.23,A -85,B 0,C 180,E1 -9270.23,E2 -9270.23} C_VEL
LIN {X 0,Y 435.74,Z 392.966,A -85,B 0,C 180,E1 -9271.443,E2 -9271.443} C_VEL
LIN {X 0,Y 434.776,Z 403.821,A -85,B 0,C 180,E1 -9272.779,E2 -9272.779} C_VEL
LIN {X 0,Y 433.895,Z 413.439,A -85,B 0,C 180,E1 -9274.18,E2 -9274.18} C_VEL
LIN {X 0,Y 433.131,Z 422.883,A -85,B 0,C 180,E1 -9275.82,E2 -9275.82} C_VEL
LIN {X 0,Y 432.476,Z 431.19,A -85,B 0,C 180,E1 -9277.565,E2 -9277.565} C_VEL
LIN {X 0,Y 431.91,Z 438.192,A -85,B 0,C 180,E1 -9279.364,E2 -9279.364} C_VEL
LIN {X 0,Y 431.572,Z 444.07,A -85,B 0,C 180,E1 -9281.269,E2 -9281.269} C_VEL
LIN {X 0,Y 431.33,Z 448.572,A -85,B 0,C 180,E1 -9283.186,E2 -9283.186} C_VEL
LIN {X 0,Y 431.154,Z 451.787,A -85,B 0,C 180,E1 -9285.118,E2 -9285.118} C_VEL
LIN {X 0,Y 431.065,Z 453.757,A -85,B 0,C 180,E1 -9287.065,E2 -9287.065} C_VEL
LIN {X 0,Y 431.097,Z 454.46,A -85,B 0,C 180,E1 -9289.029,E2 -9289.029} C_VEL
LIN {X 0,Y 431.086,Z 453.9,A -85,B 0,C 180,E1 -9291.018,E2 -9291.018} C_VEL
LIN {X 0,Y 431.154,Z 452.034,A -85,B 0,C 180,E1 -9293.03,E2 -9293.03} C_VEL
LIN {X 0,Y 431.367,Z 448.776,A -85,B 0,C 180,E1 -9295.062,E2 -9295.062} C_VEL
LIN {X 0,Y 431.589,Z 445.851,A -85,B 0,C 180,E1 -9296.411,E2 -9296.411} C_VEL
LIN {X 0,Y 431.954,Z 439.841,A -85,B 0,C 180,E1 -9298.526,E2 -9298.526} C_VEL
LIN {X 0,Y 432.561,Z 432.336,A -85,B 0,C 180,E1 -9300.557,E2 -9300.557} C_VEL
LIN {X 0,Y 433.295,Z 424.041,A -85,B 0,C 180,E1 -9302.361,E2 -9302.361} C_VEL
LIN {X 0,Y 434.182,Z 415.226,A -85,B 0,C 180,E1 -9303.948,E2 -9303.948} C_VEL
LIN {X 0,Y 435.184,Z 404.579,A -85,B 0,C 180,E1 -9305.548,E2 -9305.548} C_VEL
LIN {X 0,Y 436.315,Z 394.056,A -85,B 0,C 180,E1 -9306.87,E2 -9306.87} C_VEL
LIN {X 0,Y 437.471,Z 381.415,A -85,B 0,C 180,E1 -9308.199,E2 -9308.199} C_VEL
LIN {X 0,Y 438.602,Z 369.105,A -85,B 0,C 180,E1 -9309.267,E2 -9309.267} C_VEL
LIN {X 0,Y 439.779,Z 354.82,A -85,B 0,C 180,E1 -9310.272,E2 -9310.272} C_VEL
LIN {X 0,Y 440.725,Z 340.764,A -85,B 0,C 180,E1 -9311.053,E2 -9311.053} C_VEL
LIN {X 0,Y 441.471,Z 325.287,A -85,B 0,C 180,E1 -9311.706,E2 -9311.706} C_VEL
LIN {X 0,Y 442.116,Z 309.563,A -85,B 0,C 180,E1 -9312.153,E2 -9312.153} C_VEL
LIN {X 0,Y 444.593,Z 170.213,A -85,B 0,C 180,E1 -9314.534,E2 -9314.534} C_VEL
LIN {X 0,Y 442.121,Z 159.882,A -85,B 0,C 180,E1 -9314.897,E2 -9314.897} C_VEL
LIN {X 0,Y 435.552,Z 145.118,A -85,B 0,C 180,E1 -9315.657,E2 -9315.657} C_VEL
LIN {X 0,Y 432.357,Z 132.257,A -85,B 0,C 180,E1 -9318.494,E2 -9318.494} C_VEL
LIN {X 0,Y 432.331,Z 132.26,A -85,B 0,C 180,E1 -9321.849,E2 -9321.849} C_VEL
LIN {X 0,Y 432.34,Z 132.249,A -85,B 0,C 180,E1 -9325.322,E2 -9325.322} C_VEL
LIN {X 0,Y 432.322,Z 132.254,A -85,B 0,C 180,E1 -9328.653,E2 -9328.653} C_VEL
LIN {X 0,Y 432.348,Z 132.246,A -85,B 0,C 180,E1 -9331.874,E2 -9331.874} C_VEL
LIN {X 0,Y 432.378,Z 132.242,A -85,B 0,C 180,E1 -9335.538,E2 -9335.538} C_VEL
LIN {X 0,Y 432.351,Z 132.252,A -85,B 0,C 180,E1 -9339.046,E2 -9339.046} C_VEL
LIN {X 0,Y 432.36,Z 132.252,A -85,B 0,C 180,E1 -9342.01,E2 -9342.01} C_VEL
LIN {X 0,Y 432.394,Z 132.244,A -85,B 0,C 180,E1 -9344.926,E2 -9344.926} C_VEL
LIN {X 0,Y 432.46,Z 132.239,A -85,B 0,C 180,E1 -9347.803,E2 -9347.803} C_VEL
LIN {X 0,Y 432.492,Z 132.235,A -85,B 0,C 180,E1 -9351.59,E2 -9351.59} C_VEL
LIN {X 0,Y 432.594,Z 132.217,A -85,B 0,C 180,E1 -9354.406,E2 -9354.406} C_VEL
LIN {X 0,Y 432.603,Z 132.217,A -85,B 0,C 180,E1 -9358.138,E2 -9358.138} C_VEL
LIN {X 0,Y 432.732,Z 132.205,A -85,B 0,C 180,E1 -9360,E2 -9360} C_VEL
LIN {X 0,Y 432.592,Z 132.221,A -85,B 0,C 180,E1 -9362.793,E2 -9362.793} C_VEL
LIN {X 0,Y 432.586,Z 132.223,A -85,B 0,C 180,E1 -9365.594,E2 -9365.594} C_VEL
LIN {X 0,Y 432.463,Z 132.236,A -85,B 0,C 180,E1 -9368.41,E2 -9368.41} C_VEL
LIN {X 0,Y 432.459,Z 132.235,A -85,B 0,C 180,E1 -9372.196,E2 -9372.196} C_VEL
LIN {X 0,Y 432.43,Z 132.237,A -85,B 0,C 180,E1 -9376.039,E2 -9376.039} C_VEL
LIN {X 0,Y 432.385,Z 132.244,A -85,B 0,C 180,E1 -9379.485,E2 -9379.485} C_VEL
LIN {X 0,Y 432.318,Z 132.256,A -85,B 0,C 180,E1 -9382.964,E2 -9382.964} C_VEL
LIN {X 0,Y 432.361,Z 132.249,A -85,B 0,C 180,E1 -9386.032,E2 -9386.032} C_VEL
LIN {X 0,Y 432.341,Z 132.251,A -85,B 0,C 180,E1 -9389.187,E2 -9389.187} C_VEL
LIN {X 0,Y 432.321,Z 132.257,A -85,B 0,C 180,E1 -9392.443,E2 -9392.443} C_VEL
LIN {X 0,Y 432.341,Z 132.253,A -85,B 0,C 180,E1 -9395.631,E2 -9395.631} C_VEL
LIN {X 0,Y 432.339,Z 132.244,A -85,B 0,C 180,E1 -9398.714,E2 -9398.714} C_VEL
LIN {X 0,Y 432.332,Z 132.257,A -85,B 0,C 180,E1 -9401.797,E2 -9401.797} C_VEL
LIN {X 0,Y 432.332,Z 132.255,A -85,B 0,C 180,E1 -9404.347,E2 -9404.347} C_VEL
LIN {X 0,Y 432.318,Z 132.251,A -85,B 0,C 180,E1 -9407.016,E2 -9407.016} C_VEL
LIN {X 0,Y 432.335,Z 132.252,A -85,B 0,C 180,E1 -9409.82,E2 -9409.82} C_VEL
LIN {X 0,Y 432.305,Z 132.256,A -85,B 0,C 180,E1 -9413.022,E2 -9413.022} C_VEL
LIN {X 0,Y 432.357,Z 132.256,A -85,B 0,C 180,E1 -9415.997,E2 -9415.997} C_VEL
LIN {X 0,Y 432.372,Z 132.441,A -85,B 0,C 180,E1 -9417.285,E2 -9417.285} C_VEL
LIN {X 0,Y 436.017,Z 145.948,A -85,B 0,C 180,E1 -9420.022,E2 -9420.022} C_VEL
LIN {X 0,Y 438.459,Z 156.916,A -85,B 0,C 180,E1 -9422.106,E2 -9422.106} C_VEL
LIN {X 0,Y 437.915,Z 165.742,A -85,B 0,C 180,E1 -9423.56,E2 -9423.56} C_VEL
LIN {X 0,Y 442.788,Z 188.824,A -85,B 0,C 180,E1 -9424.336,E2 -9424.336} C_VEL
LIN {X 0,Y 444.207,Z 197.084,A -85,B 0,C 180,E1 -9424.585,E2 -9424.585} C_VEL
LIN {X 0,Y 441.83,Z 332.978,A -85,B 0,C 180,E1 -9426.909,E2 -9426.909} C_VEL
LIN {X 0,Y 441.045,Z 348.676,A -85,B 0,C 180,E1 -9427.361,E2 -9427.361} C_VEL
LIN {X 0,Y 440.152,Z 363.913,A -85,B 0,C 180,E1 -9428.004,E2 -9428.004} C_VEL
LIN {X 0,Y 439.172,Z 377.788,A -85,B 0,C 180,E1 -9428.773,E2 -9428.773} C_VEL
LIN {X 0,Y 438.007,Z 391.093,A -85,B 0,C 180,E1 -9429.697,E2 -9429.697} C_VEL
LIN {X 0,Y 436.768,Z 404.669,A -85,B 0,C 180,E1 -9430.862,E2 -9430.862} C_VEL
LIN {X 0,Y 435.485,Z 417.525,A -85,B 0,C 180,E1 -9432.206,E2 -9432.206} C_VEL
LIN {X 0,Y 434.494,Z 428.279,A -85,B 0,C 180,E1 -9433.557,E2 -9433.557} C_VEL
LIN {X 0,Y 433.463,Z 439.277,A -85,B 0,C 180,E1 -9435.205,E2 -9435.205} C_VEL
LIN {X 0,Y 432.646,Z 448.404,A -85,B 0,C 180,E1 -9436.855,E2 -9436.855} C_VEL
LIN {X 0,Y 432.081,Z 457.015,A -85,B 0,C 180,E1 -9438.745,E2 -9438.745} C_VEL
LIN {X 0,Y 431.579,Z 463.931,A -85,B 0,C 180,E1 -9440.628,E2 -9440.628} C_VEL
LIN {X 0,Y 431.342,Z 469.37,A -85,B 0,C 180,E1 -9442.511,E2 -9442.511} C_VEL
LIN {X 0,Y 431.222,Z 473.479,A -85,B 0,C 180,E1 -9444.389,E2 -9444.389} C_VEL
LIN {X 0,Y 431.137,Z 476.349,A -85,B 0,C 180,E1 -9446.262,E2 -9446.262} C_VEL
LIN {X 0,Y 431.198,Z 478.047,A -85,B 0,C 180,E1 -9448.132,E2 -9448.132} C_VEL
LIN {X 0,Y 431.164,Z 478.6,A -85,B 0,C 180,E1 -9450,E2 -9450} C_VEL
LIN {X 0,Y 431.198,Z 477.971,A -85,B 0,C 180,E1 -9451.868,E2 -9451.868} C_VEL
LIN {X 0,Y 431.139,Z 476.158,A -85,B 0,C 180,E1 -9453.739,E2 -9453.739} C_VEL
LIN {X 0,Y 431.232,Z 473.161,A -85,B 0,C 180,E1 -9455.612,E2 -9455.612} C_VEL
LIN {X 0,Y 431.379,Z 468.904,A -85,B 0,C 180,E1 -9457.489,E2 -9457.489} C_VEL
LIN {X 0,Y 431.569,Z 463.267,A -85,B 0,C 180,E1 -9459.373,E2 -9459.373} C_VEL
LIN {X 0,Y 432.064,Z 456.103,A -85,B 0,C 180,E1 -9461.256,E2 -9461.256} C_VEL
LIN {X 0,Y 432.413,Z 449.044,A -85,B 0,C 180,E1 -9462.793,E2 -9462.793} C_VEL
LIN {X 0,Y 433.221,Z 439.182,A -85,B 0,C 180,E1 -9464.564,E2 -9464.564} C_VEL
LIN {X 0,Y 433.979,Z 429.741,A -85,B 0,C 180,E1 -9465.981,E2 -9465.981} C_VEL
LIN {X 0,Y 435.052,Z 417.718,A -85,B 0,C 180,E1 -9467.492,E2 -9467.492} C_VEL
LIN {X 0,Y 436.096,Z 405.103,A -85,B 0,C 180,E1 -9468.803,E2 -9468.803} C_VEL
LIN {X 0,Y 437.283,Z 391.342,A -85,B 0,C 180,E1 -9469.971,E2 -9469.971} C_VEL
LIN {X 0,Y 438.337,Z 377.825,A -85,B 0,C 180,E1 -9470.901,E2 -9470.901} C_VEL
LIN {X 0,Y 439.255,Z 363.795,A -85,B 0,C 180,E1 -9471.668,E2 -9471.668} C_VEL
LIN {X 0,Y 440.027,Z 348.568,A -85,B 0,C 180,E1 -9472.301,E2 -9472.301} C_VEL
LIN {X 0,Y 440.701,Z 332.638,A -85,B 0,C 180,E1 -9472.751,E2 -9472.751} C_VEL
LIN {X 0,Y 442.831,Z 196.702,A -85,B 0,C 180,E1 -9475.029,E2 -9475.029} C_VEL
LIN {X 0,Y 437.117,Z 166.213,A -85,B 0,C 180,E1 -9475.895,E2 -9475.895} C_VEL
LIN {X 0,Y 437.782,Z 156.15,A -85,B 0,C 180,E1 -9477.487,E2 -9477.487} C_VEL
LIN {X 0,Y 436.194,Z 148.078,A -85,B 0,C 180,E1 -9478.906,E2 -9478.906} C_VEL
LIN {X 0,Y 432.339,Z 132.26,A -85,B 0,C 180,E1 -9481.824,E2 -9481.824} C_VEL
LIN {X 0,Y 432.341,Z 132.26,A -85,B 0,C 180,E1 -9484.678,E2 -9484.678} C_VEL
LIN {X 0,Y 432.343,Z 132.255,A -85,B 0,C 180,E1 -9488.15,E2 -9488.15} C_VEL
LIN {X 0,Y 432.326,Z 132.26,A -85,B 0,C 180,E1 -9491.601,E2 -9491.601} C_VEL
LIN {X 0,Y 432.335,Z 132.257,A -85,B 0,C 180,E1 -9494.348,E2 -9494.348} C_VEL
LIN {X 0,Y 432.322,Z 132.26,A -85,B 0,C 180,E1 -9497.016,E2 -9497.016} C_VEL
LIN {X 0,Y 432.336,Z 132.254,A -85,B 0,C 180,E1 -9499.821,E2 -9499.821} C_VEL
LIN {X 0,Y 432.308,Z 132.259,A -85,B 0,C 180,E1 -9503.023,E2 -9503.023} C_VEL
LIN {X 0,Y 432.36,Z 132.251,A -85,B 0,C 180,E1 -9505.997,E2 -9505.997} C_VEL
LIN {X 0,Y 432.349,Z 132.253,A -85,B 0,C 180,E1 -9509.491,E2 -9509.491} C_VEL
LIN {X 0,Y 432.338,Z 132.239,A -85,B 0,C 180,E1 -9511.874,E2 -9511.874} C_VEL
LIN {X 0,Y 432.381,Z 132.248,A -85,B 0,C 180,E1 -9515.539,E2 -9515.539} C_VEL
LIN {X 0,Y 432.354,Z 132.253,A -85,B 0,C 180,E1 -9519.047,E2 -9519.047} C_VEL
LIN {X 0,Y 432.363,Z 132.249,A -85,B 0,C 180,E1 -9522.011,E2 -9522.011} C_VEL
LIN {X 0,Y 432.395,Z 132.25,A -85,B 0,C 180,E1 -9524.927,E2 -9524.927} C_VEL
LIN {X 0,Y 432.464,Z 132.234,A -85,B 0,C 180,E1 -9527.804,E2 -9527.804} C_VEL
LIN {X 0,Y 432.468,Z 132.235,A -85,B 0,C 180,E1 -9531.59,E2 -9531.59} C_VEL
LIN {X 0,Y 432.575,Z 132.23,A -85,B 0,C 180,E1 -9534.406,E2 -9534.406} C_VEL
LIN {X 0,Y 432.6,Z 132.211,A -85,B 0,C 180,E1 -9538.138,E2 -9538.138} C_VEL
LIN {X 0,Y 432.624,Z 132.201,A -85,B 0,C 180,E1 -9540,E2 -9540} C_VEL
LIN {X 0,Y 432.56,Z 132.223,A -85,B 0,C 180,E1 -9542.794,E2 -9542.794} C_VEL
LIN {X 0,Y 432.519,Z 132.225,A -85,B 0,C 180,E1 -9546.532,E2 -9546.532} C_VEL
LIN {X 0,Y 432.423,Z 132.225,A -85,B 0,C 180,E1 -9549.354,E2 -9549.354} C_VEL
LIN {X 0,Y 432.423,Z 132.239,A -85,B 0,C 180,E1 -9552.796,E2 -9552.796} C_VEL
LIN {X 0,Y 432.36,Z 132.246,A -85,B 0,C 180,E1 -9556.453,E2 -9556.453} C_VEL
LIN {X 0,Y 432.296,Z 132.26,A -85,B 0,C 180,E1 -9559.963,E2 -9559.963} C_VEL
LIN {X 0,Y 432.302,Z 132.255,A -85,B 0,C 180,E1 -9562.966,E2 -9562.966} C_VEL
LIN {X 0,Y 432.309,Z 132.255,A -85,B 0,C 180,E1 -9566.037,E2 -9566.037} C_VEL
LIN {X 0,Y 432.319,Z 132.241,A -85,B 0,C 180,E1 -9569.19,E2 -9569.19} C_VEL
LIN {X 0,Y 432.309,Z 132.253,A -85,B 0,C 180,E1 -9572.445,E2 -9572.445} C_VEL
LIN {X 0,Y 432.336,Z 132.249,A -85,B 0,C 180,E1 -9575.819,E2 -9575.819} C_VEL
LIN {X 0,Y 432.304,Z 132.252,A -85,B 0,C 180,E1 -9579.348,E2 -9579.348} C_VEL
LIN {X 0,Y 432.308,Z 132.256,A -85,B 0,C 180,E1 -9581.801,E2 -9581.801} C_VEL
LIN {X 0,Y 432.337,Z 132.252,A -85,B 0,C 180,E1 -9584.348,E2 -9584.348} C_VEL
LIN {X 0,Y 432.307,Z 132.255,A -85,B 0,C 180,E1 -9587.018,E2 -9587.018} C_VEL
LIN {X 0,Y 432.293,Z 132.259,A -85,B 0,C 180,E1 -9589.828,E2 -9589.828} C_VEL
LIN {X 0,Y 432.308,Z 132.256,A -85,B 0,C 180,E1 -9593.021,E2 -9593.021} C_VEL
LIN {X 0,Y 432.338,Z 132.255,A -85,B 0,C 180,E1 -9596.002,E2 -9596.002} C_VEL
LIN {X 0,Y 432.351,Z 132.253,A -85,B 0,C 180,E1 -9599.49,E2 -9599.49} C_VEL
LIN {X 0,Y 432.333,Z 132.254,A -85,B 0,C 180,E1 -9601.873,E2 -9601.873} C_VEL
LIN {X 0,Y 432.359,Z 132.254,A -85,B 0,C 180,E1 -9605.546,E2 -9605.546} C_VEL
LIN {X 0,Y 432.355,Z 132.252,A -85,B 0,C 180,E1 -9609.046,E2 -9609.046} C_VEL
LIN {X 0,Y 432.363,Z 132.242,A -85,B 0,C 180,E1 -9612.01,E2 -9612.01} C_VEL
LIN {X 0,Y 432.398,Z 132.247,A -85,B 0,C 180,E1 -9614.926,E2 -9614.926} C_VEL
LIN {X 0,Y 432.465,Z 132.244,A -85,B 0,C 180,E1 -9617.803,E2 -9617.803} C_VEL
LIN {X 0,Y 432.449,Z 132.289,A -85,B 0,C 180,E1 -9620.588,E2 -9620.588} C_VEL
LIN {X 0,Y 435.307,Z 144.795,A -85,B 0,C 180,E1 -9623.084,E2 -9623.084} C_VEL
LIN {X 0,Y 440.449,Z 157.978,A -85,B 0,C 180,E1 -9623.614,E2 -9623.614} C_VEL
LIN {X 0,Y 443.056,Z 169.496,A -85,B 0,C 180,E1 -9623.962,E2 -9623.962} C_VEL
LIN {X 0,Y 442.538,Z 205.77,A -85,B 0,C 180,E1 -9624.569,E2 -9624.569} C_VEL
LIN {X 0,Y 441.938,Z 211.618,A -85,B 0,C 180,E1 -9624.639,E2 -9624.639} C_VEL
LIN {X 0,Y 439.101,Z 221.132,A -85,B 0,C 180,E1 -9624.654,E2 -9624.654} C_VEL
LIN {X 0,Y 436.212,Z 230.648,A -85,B 0,C 180,E1 -9624.667,E2 -9624.667} C_VEL
LIN {X 0,Y 435.534,Z 236.503,A -85,B 0,C 180,E1 -9624.734,E2 -9624.734} C_VEL
LIN {X 0,Y 434.289,Z 310.157,A -85,B 0,C 180,E1 -9625.998,E2 -9625.998} C_VEL
LIN {X 0,Y 433.729,Z 325.078,A -85,B 0,C 180,E1 -9626.429,E2 -9626.429} C_VEL
LIN {X 0,Y 432.948,Z 340.82,A -85,B 0,C 180,E1 -9627.092,E2 -9627.092} C_VEL
LIN {X 0,Y 432.07,Z 355.233,A -85,B 0,C 180,E1 -9627.902,E2 -9627.902} C_VEL
LIN {X 0,Y 431.037,Z 368.435,A -85,B 0,C 180,E1 -9628.832,E2 -9628.832} C_VEL
LIN {X 0,Y 429.892,Z 381.893,A -85,B 0,C 180,E1 -9630,E2 -9630} C_VEL
LIN {X 0,Y 428.819,Z 393.995,A -85,B 0,C 180,E1 -9631.278,E2 -9631.278} C_VEL
LIN {X 0,Y 427.86,Z 404.361,A -85,B 0,C 180,E1 -9632.589,E2 -9632.589} C_VEL
LIN {X 0,Y 426.919,Z 413.93,A -85,B 0,C 180,E1 -9634.012,E2 -9634.012} C_VEL
LIN {X 0,Y 426.121,Z 423.324,A -85,B 0,C 180,E1 -9635.679,E2 -9635.679} C_VEL
LIN {X 0,Y 425.533,Z 430.142,A -85,B 0,C 180,E1 -9637.108,E2 -9637.108} C_VEL
LIN {X 0,Y 424.911,Z 437.736,A -85,B 0,C 180,E1 -9639.04,E2 -9639.04} C_VEL
LIN {X 0,Y 424.542,Z 443.761,A -85,B 0,C 180,E1 -9640.974,E2 -9640.974} C_VEL
LIN {X 0,Y 424.351,Z 447.331,A -85,B 0,C 180,E1 -9642.433,E2 -9642.433} C_VEL
LIN {X 0,Y 424.094,Z 450.984,A -85,B 0,C 180,E1 -9644.393,E2 -9644.393} C_VEL
LIN {X 0,Y 424.015,Z 453.375,A -85,B 0,C 180,E1 -9646.366,E2 -9646.366} C_VEL
LIN {X 0,Y 423.974,Z 454.537,A -85,B 0,C 180,E1 -9648.358,E2 -9648.358} C_VEL
LIN {X 0,Y 423.966,Z 454.449,A -85,B 0,C 180,E1 -9650.372,E2 -9650.372} C_VEL
LIN {X 0,Y 424.047,Z 453.067,A -85,B 0,C 180,E1 -9652.407,E2 -9652.407} C_VEL
LIN {X 0,Y 424.193,Z 450.312,A -85,B 0,C 180,E1 -9654.469,E2 -9654.469} C_VEL
LIN {X 0,Y 424.54,Z 446.086,A -85,B 0,C 180,E1 -9656.549,E2 -9656.549} C_VEL
LIN {X 0,Y 424.916,Z 440.212,A -85,B 0,C 180,E1 -9658.662,E2 -9658.662} C_VEL
LIN {X 0,Y 425.501,Z 433.593,A -85,B 0,C 180,E1 -9660.524,E2 -9660.524} C_VEL
LIN {X 0,Y 426.294,Z 425.331,A -85,B 0,C 180,E1 -9662.398,E2 -9662.398} C_VEL
LIN {X 0,Y 427.179,Z 416.723,A -85,B 0,C 180,E1 -9664.012,E2 -9664.012} C_VEL
LIN {X 0,Y 428.249,Z 406.372,A -85,B 0,C 180,E1 -9665.633,E2 -9665.633} C_VEL
LIN {X 0,Y 429.445,Z 395.534,A -85,B 0,C 180,E1 -9667.043,E2 -9667.043} C_VEL
LIN {X 0,Y 430.642,Z 383.771,A -85,B 0,C 180,E1 -9668.327,E2 -9668.327} C_VEL
LIN {X 0,Y 431.907,Z 370.485,A -85,B 0,C 180,E1 -9669.527,E2 -9669.527} C_VEL
LIN {X 0,Y 433.047,Z 357.51,A -85,B 0,C 180,E1 -9670.479,E2 -9670.479} C_VEL
LIN {X 0,Y 434.029,Z 343.812,A -85,B 0,C 180,E1 -9671.288,E2 -9671.288} C_VEL
LIN {X 0,Y 434.89,Z 328.55,A -85,B 0,C 180,E1 -9671.979,E2 -9671.979} C_VEL
LIN {X 0,Y 435.586,Z 313.506,A -85,B 0,C 180,E1 -9672.457,E2 -9672.457} C_VEL
LIN {X 0,Y 436.072,Z 292.439,A -85,B 0,C 180,E1 -9672.87,E2 -9672.87} C_VEL
LIN {X 0,Y 438.331,Z 171.373,A -85,B 0,C 180,E1 -9674.953,E2 -9674.953} C_VEL
LIN {X 0,Y 436.09,Z 162.368,A -85,B 0,C 180,E1 -9675.283,E2 -9675.283} C_VEL
LIN {X 0,Y 429.671,Z 148.221,A -85,B 0,C 180,E1 -9676.033,E2 -9676.033} C_VEL
LIN {X 0,Y 428.379,Z 145.302,A -85,B 0,C 180,E1 -9676.208,E2 -9676.208} C_VEL
LIN {X 0,Y 425.299,Z 133.141,A -85,B 0,C 180,E1 -9678.977,E2 -9678.977} C_VEL
LIN {X 0,Y 425.277,Z 133.135,A -85,B 0,C 180,E1 -9682.488,E2 -9682.488} C_VEL
LIN {X 0,Y 425.308,Z 133.127,A -85,B 0,C 180,E1 -9685.817,E2 -9685.817} C_VEL
LIN {X 0,Y 425.291,Z 133.132,A -85,B 0,C 180,E1 -9689.239,E2 -9689.239} C_VEL
LIN {X 0,Y 425.3,Z 133.127,A -85,B 0,C 180,E1 -9692.438,E2 -9692.438} C_VEL
LIN {X 0,Y 425.346,Z 133.117,A -85,B 0,C 180,E1 -9695.601,E2 -9695.601} C_VEL
LIN {X 0,Y 425.294,Z 133.132,A -85,B 0,C 180,E1 -9698.681,E2 -9698.681} C_VEL
LIN {X 0,Y 425.322,Z 133.13,A -85,B 0,C 180,E1 -9701.702,E2 -9701.702} C_VEL
LIN {X 0,Y 425.347,Z 133.122,A -85,B 0,C 180,E1 -9704.67,E2 -9704.67} C_VEL
LIN {X 0,Y 425.413,Z 133.118,A -85,B 0,C 180,E1 -9707.598,E2 -9707.598} C_VEL
LIN {X 0,Y 425.443,Z 133.112,A -85,B 0,C 180,E1 -9711.45,E2 -9711.45} C_VEL
LIN {X 0,Y 425.551,Z 133.094,A -85,B 0,C 180,E1 -9714.313,E2 -9714.313} C_VEL
LIN {X 0,Y 425.572,Z 133.093,A -85,B 0,C 180,E1 -9718.107,E2 -9718.107} C_VEL
LIN {X 0,Y 425.702,Z 133.081,A -85,B 0,C 180,E1 -9720,E2 -9720} C_VEL
LIN {X 0,Y 425.545,Z 133.1,A -85,B 0,C 180,E1 -9722.84,E2 -9722.84} C_VEL
LIN {X 0,Y 425.541,Z 133.101,A -85,B 0,C 180,E1 -9725.687,E2 -9725.687} C_VEL
LIN {X 0,Y 425.407,Z 133.116,A -85,B 0,C 180,E1 -9728.55,E2 -9728.55} C_VEL
LIN {X 0,Y 425.412,Z 133.114,A -85,B 0,C 180,E1 -9732.401,E2 -9732.401} C_VEL
LIN {X 0,Y 425.387,Z 133.115,A -85,B 0,C 180,E1 -9736.311,E2 -9736.311} C_VEL
LIN {X 0,Y 425.327,Z 133.123,A -85,B 0,C 180,E1 -9739.635,E2 -9739.635} C_VEL
LIN {X 0,Y 425.305,Z 133.13,A -85,B 0,C 180,E1 -9743.365,E2 -9743.365} C_VEL
LIN {X 0,Y 425.346,Z 133.126,A -85,B 0,C 180,E1 -9746.844,E2 -9746.844} C_VEL
LIN {X 0,Y 425.289,Z 133.129,A -85,B 0,C 180,E1 -9749.719,E2 -9749.719} C_VEL
LIN {X 0,Y 425.28,Z 133.136,A -85,B 0,C 180,E1 -9753.048,E2 -9753.048} C_VEL
LIN {X 0,Y 425.28,Z 133.134,A -85,B 0,C 180,E1 -9755.928,E2 -9755.928} C_VEL
LIN {X 0,Y 425.286,Z 133.123,A -85,B 0,C 180,E1 -9759.042,E2 -9759.042} C_VEL
LIN {X 0,Y 425.289,Z 133.132,A -85,B 0,C 180,E1 -9761.958,E2 -9761.958} C_VEL
LIN {X 0,Y 425.283,Z 133.134,A -85,B 0,C 180,E1 -9765.283,E2 -9765.283} C_VEL
LIN {X 0,Y 425.273,Z 133.137,A -85,B 0,C 180,E1 -9768.622,E2 -9768.622} C_VEL
LIN {X 0,Y 425.308,Z 133.133,A -85,B 0,C 180,E1 -9771.103,E2 -9771.103} C_VEL
LIN {X 0,Y 425.298,Z 133.13,A -85,B 0,C 180,E1 -9774.664,E2 -9774.664} C_VEL
LIN {X 0,Y 425.321,Z 133.234,A -85,B 0,C 180,E1 -9776.779,E2 -9776.779} C_VEL
LIN {X 0,Y 429.086,Z 147.233,A -85,B 0,C 180,E1 -9779.688,E2 -9779.688} C_VEL
LIN {X 0,Y 431.595,Z 158.173,A -85,B 0,C 180,E1 -9781.821,E2 -9781.821} C_VEL
LIN {X 0,Y 431.684,Z 161.211,A -85,B 0,C 180,E1 -9782.355,E2 -9782.355} C_VEL
LIN {X 0,Y 431.313,Z 165.702,A -85,B 0,C 180,E1 -9783.082,E2 -9783.082} C_VEL
LIN {X 0,Y 436.111,Z 187.782,A -85,B 0,C 180,E1 -9783.849,E2 -9783.849} C_VEL
LIN {X 0,Y 437.937,Z 198.164,A -85,B 0,C 180,E1 -9784.172,E2 -9784.172} C_VEL
LIN {X 0,Y 435.43,Z 331.765,A -85,B 0,C 180,E1 -9786.486,E2 -9786.486} C_VEL
LIN {X 0,Y 434.688,Z 347.838,A -85,B 0,C 180,E1 -9786.948,E2 -9786.948} C_VEL
LIN {X 0,Y 433.787,Z 362.428,A -85,B 0,C 180,E1 -9787.557,E2 -9787.557} C_VEL
LIN {X 0,Y 432.69,Z 376.229,A -85,B 0,C 180,E1 -9788.314,E2 -9788.314} C_VEL
LIN {X 0,Y 431.508,Z 389.776,A -85,B 0,C 180,E1 -9789.253,E2 -9789.253} C_VEL
LIN {X 0,Y 430.273,Z 402.274,A -85,B 0,C 180,E1 -9790.313,E2 -9790.313} C_VEL
LIN {X 0,Y 428.981,Z 414.98,A -85,B 0,C 180,E1 -9791.617,E2 -9791.617} C_VEL
LIN {X 0,Y 427.817,Z 426.537,A -85,B 0,C 180,E1 -9793.047,E2 -9793.047} C_VEL
LIN {X 0,Y 426.814,Z 436.286,A -85,B 0,C 180,E1 -9794.48,E2 -9794.48} C_VEL
LIN {X 0,Y 425.859,Z 445.868,A -85,B 0,C 180,E1 -9796.155,E2 -9796.155} C_VEL
LIN {X 0,Y 425.199,Z 453.886,A -85,B 0,C 180,E1 -9797.835,E2 -9797.835} C_VEL
LIN {X 0,Y 424.71,Z 460.566,A -85,B 0,C 180,E1 -9799.513,E2 -9799.513} C_VEL
LIN {X 0,Y 424.384,Z 466.706,A -85,B 0,C 180,E1 -9801.429,E2 -9801.429} C_VEL
LIN {X 0,Y 424.21,Z 471.446,A -85,B 0,C 180,E1 -9803.341,E2 -9803.341} C_VEL
LIN {X 0,Y 424.113,Z 474.906,A -85,B 0,C 180,E1 -9805.248,E2 -9805.248} C_VEL
LIN {X 0,Y 424.11,Z 477.166,A -85,B 0,C 180,E1 -9807.151,E2 -9807.151} C_VEL
LIN {X 0,Y 424.085,Z 478.27,A -85,B 0,C 180,E1 -9809.051,E2 -9809.051} C_VEL
LIN {X 0,Y 424.085,Z 478.233,A -85,B 0,C 180,E1 -9810.95,E2 -9810.95} C_VEL
LIN {X 0,Y 424.112,Z 476.99,A -85,B 0,C 180,E1 -9812.85,E2 -9812.85} C_VEL
LIN {X 0,Y 424.137,Z 474.572,A -85,B 0,C 180,E1 -9814.753,E2 -9814.753} C_VEL
LIN {X 0,Y 424.237,Z 470.934,A -85,B 0,C 180,E1 -9816.66,E2 -9816.66} C_VEL
LIN {X 0,Y 424.374,Z 465.976,A -85,B 0,C 180,E1 -9818.572,E2 -9818.572} C_VEL
LIN {X 0,Y 424.689,Z 459.569,A -85,B 0,C 180,E1 -9820.489,E2 -9820.489} C_VEL
LIN {X 0,Y 425.198,Z 452.662,A -85,B 0,C 180,E1 -9822.166,E2 -9822.166} C_VEL
LIN {X 0,Y 425.764,Z 444.316,A -85,B 0,C 180,E1 -9823.849,E2 -9823.849} C_VEL
LIN {X 0,Y 426.62,Z 434.261,A -85,B 0,C 180,E1 -9825.528,E2 -9825.528} C_VEL
LIN {X 0,Y 427.612,Z 423.957,A -85,B 0,C 180,E1 -9826.962,E2 -9826.962} C_VEL
LIN {X 0,Y 428.682,Z 411.68,A -85,B 0,C 180,E1 -9828.397,E2 -9828.397} C_VEL
LIN {X 0,Y 429.814,Z 399.353,A -85,B 0,C 180,E1 -9829.585,E2 -9829.585} C_VEL
LIN {X 0,Y 430.883,Z 385.903,A -85,B 0,C 180,E1 -9830.654,E2 -9830.654} C_VEL
LIN {X 0,Y 432.062,Z 371.057,A -85,B 0,C 180,E1 -9831.594,E2 -9831.594} C_VEL
LIN {X 0,Y 432.972,Z 356.659,A -85,B 0,C 180,E1 -9832.298,E2 -9832.298} C_VEL
LIN {X 0,Y 433.689,Z 341.791,A -85,B 0,C 180,E1 -9832.834,E2 -9832.834} C_VEL
LIN {X 0,Y 434.193,Z 326.09,A -85,B 0,C 180,E1 -9833.206,E2 -9833.206} C_VEL
LIN {X 0,Y 436.253,Z 197.89,A -85,B 0,C 180,E1 -9835.367,E2 -9835.367} C_VEL
LIN {X 0,Y 430.366,Z 166.041,A -85,B 0,C 180,E1 -9836.284,E2 -9836.284} C_VEL
LIN {X 0,Y 430.92,Z 157.367,A -85,B 0,C 180,E1 -9837.683,E2 -9837.683} C_VEL
LIN {X 0,Y 428.033,Z 144.264,A -85,B 0,C 180,E1 -9840.052,E2 -9840.052} C_VEL
LIN {X 0,Y 425.287,Z 133.138,A -85,B 0,C 180,E1 -9842.173,E2 -9842.173} C_VEL
LIN {X 0,Y 425.301,Z 133.139,A -85,B 0,C 180,E1 -9845.336,E2 -9845.336} C_VEL
LIN {X 0,Y 425.298,Z 133.132,A -85,B 0,C 180,E1 -9848.899,E2 -9848.899} C_VEL
LIN {X 0,Y 425.284,Z 133.137,A -85,B 0,C 180,E1 -9851.958,E2 -9851.958} C_VEL
LIN {X 0,Y 425.287,Z 133.138,A -85,B 0,C 180,E1 -9855.284,E2 -9855.284} C_VEL
LIN {X 0,Y 425.276,Z 133.135,A -85,B 0,C 180,E1 -9858.622,E2 -9858.622} C_VEL
LIN {X 0,Y 425.295,Z 133.128,A -85,B 0,C 180,E1 -9861.101,E2 -9861.101} C_VEL
LIN {X 0,Y 425.301,Z 133.129,A -85,B 0,C 180,E1 -9864.665,E2 -9864.665} C_VEL
LIN {X 0,Y 425.267,Z 133.133,A -85,B 0,C 180,E1 -9868.074,E2 -9868.074} C_VEL
LIN {X 0,Y 425.308,Z 133.118,A -85,B 0,C 180,E1 -9871.367,E2 -9871.367} C_VEL
LIN {X 0,Y 425.272,Z 133.129,A -85,B 0,C 180,E1 -9874.554,E2 -9874.554} C_VEL
LIN {X 0,Y 425.307,Z 133.131,A -85,B 0,C 180,E1 -9876.635,E2 -9876.635} C_VEL
LIN {X 0,Y 425.332,Z 133.127,A -85,B 0,C 180,E1 -9880.365,E2 -9880.365} C_VEL
LIN {X 0,Y 425.392,Z 133.115,A -85,B 0,C 180,E1 -9883.689,E2 -9883.689} C_VEL
LIN {X 0,Y 425.416,Z 133.111,A -85,B 0,C 180,E1 -9887.599,E2 -9887.599} C_VEL
LIN {X 0,Y 425.412,Z 133.114,A -85,B 0,C 180,E1 -9891.45,E2 -9891.45} C_VEL
LIN {X 0,Y 425.529,Z 133.106,A -85,B 0,C 180,E1 -9894.313,E2 -9894.313} C_VEL
LIN {X 0,Y 425.569,Z 133.086,A -85,B 0,C 180,E1 -9898.108,E2 -9898.108} C_VEL
LIN {X 0,Y 425.577,Z 133.078,A -85,B 0,C 180,E1 -9900,E2 -9900} C_VEL
LIN {X 0,Y 425.515,Z 133.101,A -85,B 0,C 180,E1 -9902.841,E2 -9902.841} C_VEL
LIN {X 0,Y 425.48,Z 133.101,A -85,B 0,C 180,E1 -9906.64,E2 -9906.64} C_VEL
LIN {X 0,Y 425.384,Z 133.101,A -85,B 0,C 180,E1 -9909.51,E2 -9909.51} C_VEL
LIN {X 0,Y 425.389,Z 133.115,A -85,B 0,C 180,E1 -9912.898,E2 -9912.898} C_VEL
LIN {X 0,Y 425.317,Z 133.123,A -85,B 0,C 180,E1 -9916.582,E2 -9916.582} C_VEL
LIN {X 0,Y 425.281,Z 133.138,A -85,B 0,C 180,E1 -9919.616,E2 -9919.616} C_VEL
LIN {X 0,Y 425.288,Z 133.127,A -85,B 0,C 180,E1 -9922.339,E2 -9922.339} C_VEL
LIN {X 0,Y 425.253,Z 133.139,A -85,B 0,C 180,E1 -9925.449,E2 -9925.449} C_VEL
LIN {X 0,Y 425.3,Z 133.117,A -85,B 0,C 180,E1 -9928.857,E2 -9928.857} C_VEL
LIN {X 0,Y 425.251,Z 133.132,A -85,B 0,C 180,E1 -9931.929,E2 -9931.929} C_VEL
LIN {X 0,Y 425.295,Z 133.13,A -85,B 0,C 180,E1 -9935.337,E2 -9935.337} C_VEL
LIN {X 0,Y 425.28,Z 133.12,A -85,B 0,C 180,E1 -9938.901,E2 -9938.901} C_VEL
LIN {X 0,Y 425.261,Z 133.139,A -85,B 0,C 180,E1 -9942.655,E2 -9942.655} C_VEL
LIN {X 0,Y 425.288,Z 133.119,A -85,B 0,C 180,E1 -9945.283,E2 -9945.283} C_VEL
LIN {X 0,Y 425.253,Z 133.14,A -85,B 0,C 180,E1 -9948.618,E2 -9948.618} C_VEL
LIN {X 0,Y 425.283,Z 133.127,A -85,B 0,C 180,E1 -9951.099,E2 -9951.099} C_VEL
LIN {X 0,Y 425.3,Z 133.135,A -85,B 0,C 180,E1 -9954.664,E2 -9954.664} C_VEL
LIN {X 0,Y 425.268,Z 133.13,A -85,B 0,C 180,E1 -9958.073,E2 -9958.073} C_VEL
LIN {X 0,Y 425.31,Z 133.127,A -85,B 0,C 180,E1 -9961.366,E2 -9961.366} C_VEL
LIN {X 0,Y 425.265,Z 133.14,A -85,B 0,C 180,E1 -9964.552,E2 -9964.552} C_VEL
LIN {X 0,Y 425.297,Z 133.135,A -85,B 0,C 180,E1 -9967.729,E2 -9967.729} C_VEL
LIN {X 0,Y 425.366,Z 133.121,A -85,B 0,C 180,E1 -9970.704,E2 -9970.704} C_VEL
LIN {X 0,Y 425.393,Z 133.118,A -85,B 0,C 180,E1 -9973.688,E2 -9973.688} C_VEL
LIN {X 0,Y 425.418,Z 133.12,A -85,B 0,C 180,E1 -9977.598,E2 -9977.598} C_VEL
LIN {X 0,Y 425.42,Z 133.273,A -85,B 0,C 180,E1 -9980.281,E2 -9980.281} C_VEL
LIN {X 0,Y 428.138,Z 145.004,A -85,B 0,C 180,E1 -9982.667,E2 -9982.667} C_VEL
LIN {X 0,Y 434.307,Z 160.693,A -85,B 0,C 180,E1 -9983.312,E2 -9983.312} C_VEL
LIN {X 0,Y 436.55,Z 170.766,A -85,B 0,C 180,E1 -9983.621,E2 -9983.621} C_VEL
LIN {X 0,Y 435.534,Z 236.503,A -85,B 0,C 180,E1 -9984.734,E2 -9984.734} C_VEL
LIN {X 0,Y 434.878,Z 242.347,A -85,B 0,C 180,E1 -9984.802,E2 -9984.802} C_VEL
LIN {X 0,Y 429.161,Z 261.357,A -85,B 0,C 180,E1 -9984.833,E2 -9984.833} C_VEL
LIN {X 0,Y 428.419,Z 267.206,A -85,B 0,C 180,E1 -9984.898,E2 -9984.898} C_VEL
LIN {X 0,Y 427.651,Z 310.682,A -85,B 0,C 180,E1 -9985.67,E2 -9985.67} C_VEL
LIN {X 0,Y 427.071,Z 325.508,A -85,B 0,C 180,E1 -9986.107,E2 -9986.107} C_VEL
LIN {X 0,Y 426.301,Z 340.608,A -85,B 0,C 180,E1 -9986.751,E2 -9986.751} C_VEL
LIN {X 0,Y 425.427,Z 354.171,A -85,B 0,C 180,E1 -9987.514,E2 -9987.514} C_VEL
LIN {X 0,Y 424.237,Z 369.114,A -85,B 0,C 180,E1 -9988.576,E2 -9988.576} C_VEL
LIN {X 0,Y 423.042,Z 382.482,A -85,B 0,C 180,E1 -9989.762,E2 -9989.762} C_VEL
LIN {X 0,Y 421.904,Z 394.826,A -85,B 0,C 180,E1 -9991.097,E2 -9991.097} C_VEL
LIN {X 0,Y 420.78,Z 406.568,A -85,B 0,C 180,E1 -9992.632,E2 -9992.632} C_VEL
LIN {X 0,Y 419.838,Z 415.866,A -85,B 0,C 180,E1 -9994.079,E2 -9994.079} C_VEL
LIN {X 0,Y 419.04,Z 424.976,A -85,B 0,C 180,E1 -9995.775,E2 -9995.775} C_VEL
LIN {X 0,Y 418.322,Z 433.041,A -85,B 0,C 180,E1 -9997.59,E2 -9997.59} C_VEL
LIN {X 0,Y 417.808,Z 438.906,A -85,B 0,C 180,E1 -9999.195,E2 -9999.195} C_VEL
LIN {X 0,Y 417.434,Z 444.712,A -85,B 0,C 180,E1 -10001.164,E2 -10001.164} C_VEL
LIN {X 0,Y 417.216,Z 448.184,A -85,B 0,C 180,E1 -10002.649,E2 -10002.649} C_VEL
LIN {X 0,Y 416.986,Z 451.631,A -85,B 0,C 180,E1 -10004.644,E2 -10004.644} C_VEL
LIN {X 0,Y 416.912,Z 453.825,A -85,B 0,C 180,E1 -10006.653,E2 -10006.653} C_VEL
LIN {X 0,Y 416.88,Z 454.789,A -85,B 0,C 180,E1 -10008.682,E2 -10008.682} C_VEL
LIN {X 0,Y 416.868,Z 454.5,A -85,B 0,C 180,E1 -10010.734,E2 -10010.734} C_VEL
LIN {X 0,Y 416.974,Z 452.91,A -85,B 0,C 180,E1 -10012.809,E2 -10012.809} C_VEL
LIN {X 0,Y 417.164,Z 449.941,A -85,B 0,C 180,E1 -10014.909,E2 -10014.909} C_VEL
LIN {X 0,Y 417.489,Z 445.943,A -85,B 0,C 180,E1 -10016.848,E2 -10016.848} C_VEL
LIN {X 0,Y 417.964,Z 439.863,A -85,B 0,C 180,E1 -10019.028,E2 -10019.028} C_VEL
LIN {X 0,Y 418.504,Z 434.039,A -85,B 0,C 180,E1 -10020.693,E2 -10020.693} C_VEL
LIN {X 0,Y 419.268,Z 426.57,A -85,B 0,C 180,E1 -10022.439,E2 -10022.439} C_VEL
LIN {X 0,Y 420.166,Z 418.145,A -85,B 0,C 180,E1 -10024.079,E2 -10024.079} C_VEL
LIN {X 0,Y 421.316,Z 408.059,A -85,B 0,C 180,E1 -10025.721,E2 -10025.721} C_VEL
LIN {X 0,Y 422.541,Z 397.782,A -85,B 0,C 180,E1 -10027.118,E2 -10027.118} C_VEL
LIN {X 0,Y 423.739,Z 386.13,A -85,B 0,C 180,E1 -10028.458,E2 -10028.458} C_VEL
LIN {X 0,Y 425.075,Z 373.18,A -85,B 0,C 180,E1 -10029.688,E2 -10029.688} C_VEL
LIN {X 0,Y 426.332,Z 360.334,A -85,B 0,C 180,E1 -10030.685,E2 -10030.685} C_VEL
LIN {X 0,Y 427.356,Z 347.046,A -85,B 0,C 180,E1 -10031.525,E2 -10031.525} C_VEL
LIN {X 0,Y 428.33,Z 332.467,A -85,B 0,C 180,E1 -10032.238,E2 -10032.238} C_VEL
LIN {X 0,Y 429.07,Z 318.365,A -85,B 0,C 180,E1 -10032.744,E2 -10032.744} C_VEL
LIN {X 0,Y 429.542,Z 303.05,A -85,B 0,C 180,E1 -10033.108,E2 -10033.108} C_VEL
LIN {X 0,Y 432.106,Z 172.652,A -85,B 0,C 180,E1 -10035.381,E2 -10035.381} C_VEL
LIN {X 0,Y 430.302,Z 165.432,A -85,B 0,C 180,E1 -10035.653,E2 -10035.653} C_VEL
LIN {X 0,Y 424.117,Z 151.754,A -85,B 0,C 180,E1 -10036.403,E2 -10036.403} C_VEL
LIN {X 0,Y 421.24,Z 145.525,A -85,B 0,C 180,E1 -10036.78,E2 -10036.78} C_VEL
LIN {X 0,Y 418.253,Z 134.016,A -85,B 0,C 180,E1 -10039.492,E2 -10039.492} C_VEL
LIN {X 0,Y 418.239,Z 134.012,A -85,B 0,C 180,E1 -10042.775,E2 -10042.775} C_VEL
LIN {X 0,Y 418.25,Z 134.013,A -85,B 0,C 180,E1 -10046.322,E2 -10046.322} C_VEL
LIN {X 0,Y 418.243,Z 134.012,A -85,B 0,C 180,E1 -10049.727,E2 -10049.727} C_VEL
LIN {X 0,Y 418.262,Z 134.007,A -85,B 0,C 180,E1 -10053.02,E2 -10053.02} C_VEL
LIN {X 0,Y 418.274,Z 133.996,A -85,B 0,C 180,E1 -10056.218,E2 -10056.218} C_VEL
LIN {X 0,Y 418.251,Z 134.01,A -85,B 0,C 180,E1 -10059.337,E2 -10059.337} C_VEL
LIN {X 0,Y 418.28,Z 134.005,A -85,B 0,C 180,E1 -10062.395,E2 -10062.395} C_VEL
LIN {X 0,Y 418.302,Z 134.001,A -85,B 0,C 180,E1 -10065.403,E2 -10065.403} C_VEL
LIN {X 0,Y 418.315,Z 133.999,A -85,B 0,C 180,E1 -10068.369,E2 -10068.369} C_VEL
LIN {X 0,Y 418.514,Z 133.977,A -85,B 0,C 180,E1 -10072.279,E2 -10072.279} C_VEL
LIN {X 0,Y 418.51,Z 133.971,A -85,B 0,C 180,E1 -10074.217,E2 -10074.217} C_VEL
LIN {X 0,Y 418.541,Z 133.969,A -85,B 0,C 180,E1 -10078.075,E2 -10078.075} C_VEL
LIN {X 0,Y 418.671,Z 133.957,A -85,B 0,C 180,E1 -10080,E2 -10080} C_VEL
LIN {X 0,Y 418.5,Z 133.977,A -85,B 0,C 180,E1 -10082.887,E2 -10082.887} C_VEL
LIN {X 0,Y 418.499,Z 133.978,A -85,B 0,C 180,E1 -10085.783,E2 -10085.783} C_VEL
LIN {X 0,Y 418.377,Z 133.992,A -85,B 0,C 180,E1 -10088.695,E2 -10088.695} C_VEL
LIN {X 0,Y 418.315,Z 133.999,A -85,B 0,C 180,E1 -10091.631,E2 -10091.631} C_VEL
LIN {X 0,Y 418.302,Z 134.004,A -85,B 0,C 180,E1 -10094.597,E2 -10094.597} C_VEL
LIN {X 0,Y 418.285,Z 134.005,A -85,B 0,C 180,E1 -10097.604,E2 -10097.604} C_VEL
LIN {X 0,Y 418.249,Z 134.009,A -85,B 0,C 180,E1 -10100.663,E2 -10100.663} C_VEL
LIN {X 0,Y 418.286,Z 134.003,A -85,B 0,C 180,E1 -10103.781,E2 -10103.781} C_VEL
LIN {X 0,Y 418.309,Z 134.005,A -85,B 0,C 180,E1 -10107.07,E2 -10107.07} C_VEL
LIN {X 0,Y 418.243,Z 134.01,A -85,B 0,C 180,E1 -10110.272,E2 -10110.272} C_VEL
LIN {X 0,Y 418.246,Z 134.01,A -85,B 0,C 180,E1 -10113.677,E2 -10113.677} C_VEL
LIN {X 0,Y 418.238,Z 134.008,A -85,B 0,C 180,E1 -10117.224,E2 -10117.224} C_VEL
LIN {X 0,Y 418.245,Z 134.004,A -85,B 0,C 180,E1 -10119.682,E2 -10119.682} C_VEL
LIN {X 0,Y 418.228,Z 134.006,A -85,B 0,C 180,E1 -10122.321,E2 -10122.321} C_VEL
LIN {X 0,Y 418.234,Z 134.013,A -85,B 0,C 180,E1 -10125.109,E2 -10125.109} C_VEL
LIN {X 0,Y 418.239,Z 134.009,A -85,B 0,C 180,E1 -10127.767,E2 -10127.767} C_VEL
LIN {X 0,Y 418.254,Z 134.008,A -85,B 0,C 180,E1 -10130.619,E2 -10130.619} C_VEL
LIN {X 0,Y 418.242,Z 134.017,A -85,B 0,C 180,E1 -10133.976,E2 -10133.976} C_VEL
LIN {X 0,Y 418.284,Z 134.032,A -85,B 0,C 180,E1 -10136.254,E2 -10136.254} C_VEL
LIN {X 0,Y 421.98,Z 147.746,A -85,B 0,C 180,E1 -10139.184,E2 -10139.184} C_VEL
LIN {X 0,Y 424.792,Z 159.675,A -85,B 0,C 180,E1 -10141.569,E2 -10141.569} C_VEL
LIN {X 0,Y 424.959,Z 162.898,A -85,B 0,C 180,E1 -10142.152,E2 -10142.152} C_VEL
LIN {X 0,Y 424.723,Z 165.303,A -85,B 0,C 180,E1 -10142.558,E2 -10142.558} C_VEL
LIN {X 0,Y 429.247,Z 185.909,A -85,B 0,C 180,E1 -10143.314,E2 -10143.314} C_VEL
LIN {X 0,Y 431.68,Z 199.292,A -85,B 0,C 180,E1 -10143.747,E2 -10143.747} C_VEL
LIN {X 0,Y 429.052,Z 332.11,A -85,B 0,C 180,E1 -10146.083,E2 -10146.083} C_VEL
LIN {X 0,Y 428.246,Z 347.931,A -85,B 0,C 180,E1 -10146.549,E2 -10146.549} C_VEL
LIN {X 0,Y 427.337,Z 361.822,A -85,B 0,C 180,E1 -10147.137,E2 -10147.137} C_VEL
LIN {X 0,Y 426.115,Z 376.658,A -85,B 0,C 180,E1 -10147.962,E2 -10147.962} C_VEL
LIN {X 0,Y 424.864,Z 390.052,A -85,B 0,C 180,E1 -10148.913,E2 -10148.913} C_VEL
LIN {X 0,Y 423.459,Z 403.734,A -85,B 0,C 180,E1 -10150.109,E2 -10150.109} C_VEL
LIN {X 0,Y 422.118,Z 416.157,A -85,B 0,C 180,E1 -10151.433,E2 -10151.433} C_VEL
LIN {X 0,Y 420.995,Z 426.595,A -85,B 0,C 180,E1 -10152.764,E2 -10152.764} C_VEL
LIN {X 0,Y 419.902,Z 436.301,A -85,B 0,C 180,E1 -10154.218,E2 -10154.218} C_VEL
LIN {X 0,Y 418.905,Z 445.847,A -85,B 0,C 180,E1 -10155.921,E2 -10155.921} C_VEL
LIN {X 0,Y 418.208,Z 453.822,A -85,B 0,C 180,E1 -10157.628,E2 -10157.628} C_VEL
LIN {X 0,Y 417.691,Z 460.47,A -85,B 0,C 180,E1 -10159.334,E2 -10159.334} C_VEL
LIN {X 0,Y 417.303,Z 466.585,A -85,B 0,C 180,E1 -10161.282,E2 -10161.282} C_VEL
LIN {X 0,Y 417.139,Z 471.307,A -85,B 0,C 180,E1 -10163.227,E2 -10163.227} C_VEL
LIN {X 0,Y 417.022,Z 474.749,A -85,B 0,C 180,E1 -10165.167,E2 -10165.167} C_VEL
LIN {X 0,Y 417.005,Z 476.989,A -85,B 0,C 180,E1 -10167.102,E2 -10167.102} C_VEL
LIN {X 0,Y 417.007,Z 478.076,A -85,B 0,C 180,E1 -10169.035,E2 -10169.035} C_VEL
LIN {X 0,Y 417.007,Z 478.023,A -85,B 0,C 180,E1 -10170.966,E2 -10170.966} C_VEL
LIN {X 0,Y 417.007,Z 476.766,A -85,B 0,C 180,E1 -10172.899,E2 -10172.899} C_VEL
LIN {X 0,Y 417.044,Z 474.327,A -85,B 0,C 180,E1 -10174.834,E2 -10174.834} C_VEL
LIN {X 0,Y 417.156,Z 470.667,A -85,B 0,C 180,E1 -10176.773,E2 -10176.773} C_VEL
LIN {X 0,Y 417.292,Z 465.685,A -85,B 0,C 180,E1 -10178.719,E2 -10178.719} C_VEL
LIN {X 0,Y 417.663,Z 459.253,A -85,B 0,C 180,E1 -10180.667,E2 -10180.667} C_VEL
LIN {X 0,Y 418.232,Z 451.185,A -85,B 0,C 180,E1 -10182.619,E2 -10182.619} C_VEL
LIN {X 0,Y 418.913,Z 442.575,A -85,B 0,C 180,E1 -10184.328,E2 -10184.328} C_VEL
LIN {X 0,Y 419.853,Z 432.187,A -85,B 0,C 180,E1 -10186.034,E2 -10186.034} C_VEL
LIN {X 0,Y 420.908,Z 421.55,A -85,B 0,C 180,E1 -10187.491,E2 -10187.491} C_VEL
LIN {X 0,Y 422.001,Z 409.96,A -85,B 0,C 180,E1 -10188.825,E2 -10188.825} C_VEL
LIN {X 0,Y 423.158,Z 397.335,A -85,B 0,C 180,E1 -10190.033,E2 -10190.033} C_VEL
LIN {X 0,Y 424.318,Z 383.469,A -85,B 0,C 180,E1 -10191.116,E2 -10191.116} C_VEL
LIN {X 0,Y 425.488,Z 369.059,A -85,B 0,C 180,E1 -10192.009,E2 -10192.009} C_VEL
LIN {X 0,Y 426.403,Z 354.07,A -85,B 0,C 180,E1 -10192.726,E2 -10192.726} C_VEL
LIN {X 0,Y 427.15,Z 339.595,A -85,B 0,C 180,E1 -10193.229,E2 -10193.229} C_VEL
LIN {X 0,Y 427.589,Z 323.747,A -85,B 0,C 180,E1 -10193.586,E2 -10193.586} C_VEL
LIN {X 0,Y 429.713,Z 199.158,A -85,B 0,C 180,E1 -10195.713,E2 -10195.713} C_VEL
LIN {X 0,Y 423.625,Z 165.773,A -85,B 0,C 180,E1 -10196.701,E2 -10196.701} C_VEL
LIN {X 0,Y 424.039,Z 158.79,A -85,B 0,C 180,E1 -10197.847,E2 -10197.847} C_VEL
LIN {X 0,Y 421.042,Z 145.343,A -85,B 0,C 180,E1 -10200.327,E2 -10200.327} C_VEL
LIN {X 0,Y 418.248,Z 134.014,A -85,B 0,C 180,E1 -10202.528,E2 -10202.528} C_VEL
LIN {X 0,Y 418.261,Z 134.015,A -85,B 0,C 180,E1 -10204.842,E2 -10204.842} C_VEL
LIN {X 0,Y 418.251,Z 134.011,A -85,B 0,C 180,E1 -10208.443,E2 -10208.443} C_VEL
LIN {X 0,Y 418.221,Z 134.014,A -85,B 0,C 180,E1 -10210.949,E2 -10210.949} C_VEL
LIN {X 0,Y 418.211,Z 134.02,A -85,B 0,C 180,E1 -10213.73,E2 -10213.73} C_VEL
LIN {X 0,Y 418.211,Z 134.017,A -85,B 0,C 180,E1 -10216.449,E2 -10216.449} C_VEL
LIN {X 0,Y 418.225,Z 134.017,A -85,B 0,C 180,E1 -10219.131,E2 -10219.131} C_VEL
LIN {X 0,Y 418.227,Z 134.011,A -85,B 0,C 180,E1 -10222.168,E2 -10222.168} C_VEL
LIN {X 0,Y 418.267,Z 134.012,A -85,B 0,C 180,E1 -10225.421,E2 -10225.421} C_VEL
LIN {X 0,Y 418.213,Z 134.013,A -85,B 0,C 180,E1 -10228.604,E2 -10228.604} C_VEL
LIN {X 0,Y 418.221,Z 133.997,A -85,B 0,C 180,E1 -10231.932,E2 -10231.932} C_VEL
LIN {X 0,Y 418.276,Z 134.008,A -85,B 0,C 180,E1 -10235.162,E2 -10235.162} C_VEL
LIN {X 0,Y 418.238,Z 134.007,A -85,B 0,C 180,E1 -10238.304,E2 -10238.304} C_VEL
LIN {X 0,Y 418.279,Z 134.004,A -85,B 0,C 180,E1 -10241.383,E2 -10241.383} C_VEL
LIN {X 0,Y 418.304,Z 134.002,A -85,B 0,C 180,E1 -10244.406,E2 -10244.406} C_VEL
LIN {X 0,Y 418.36,Z 133.99,A -85,B 0,C 180,E1 -10247.386,E2 -10247.386} C_VEL
LIN {X 0,Y 418.342,Z 134.001,A -85,B 0,C 180,E1 -10250.329,E2 -10250.329} C_VEL
LIN {X 0,Y 418.445,Z 133.982,A -85,B 0,C 180,E1 -10253.249,E2 -10253.249} C_VEL
LIN {X 0,Y 418.321,Z 133.999,A -85,B 0,C 180,E1 -10255.182,E2 -10255.182} C_VEL
LIN {X 0,Y 418.538,Z 133.962,A -85,B 0,C 180,E1 -10258.076,E2 -10258.076} C_VEL
LIN {X 0,Y 418.412,Z 133.977,A -85,B 0,C 180,E1 -10260.963,E2 -10260.963} C_VEL
LIN {X 0,Y 418.472,Z 133.978,A -85,B 0,C 180,E1 -10262.888,E2 -10262.888} C_VEL
